// TIA Portal V17 program export: 11 tag tables, 0 data types, 34 data blocks, 53 code blocks (in call order from the OBs), 52 instance data blocks

VAR_GLOBAL   // PLC tag table "Default tag table"
END_VAR

VAR_GLOBAL   // PLC tag table "St0_In"
   IO_AU_1 AT %I0.0 : Bool;   // Arrêt d'urgence n°1
   IO_AU_2 AT %I0.1 : Bool;   // Arrêt d'urgence n°2
   IO_BP_Rearm AT %I0.2 : Bool;   // Réarmement machine
   IO_Barillet_MP AT %I0.3 : Bool;   // Barillet Métaux Précieux ouvert (MP)
   IO_PorteEntree_Fermee AT %I0.4 : Bool;   // Porte d'entrée : Fermée
   IO_PorteSortie_Fermee AT %I0.5 : Bool;   // Porte de sortie : Fermée
   IO_PorteVision_Fermee AT %I0.6 : Bool;   // Porte maintenance vision façade : Fermée
   IO_PorteArriere_Fermee AT %I0.7 : Bool;   // Portes maitenance arrière machine : Fermée
END_VAR

VAR_GLOBAL   // PLC tag table "St0_Out"
   IO_Verrou_PorteEntree AT %Q0.0 : Bool;   // Verrouillage : Porte d'entrée
   IO_Verrou_PorteSortie AT %Q0.1 : Bool;   // Verrouillage : Porte de sortie
   IO_Verrou_PorteVision AT %Q0.2 : Bool;   // Verrouillage : Porte maintenance vision façade
   IO_Verrou_PorteArriere AT %Q0.3 : Bool;   // Verrouillage : Porte maintenance arrière machine
   IO_Ouverture_PorteEntree AT %Q0.4 : Bool;   // Ouverture : Porte d'entrée
   IO_Ouverture_PorteSortie AT %Q0.5 : Bool;   // Ouverture : Porte de sortie
   IO_LED_Rouge AT %Q0.6 : Bool;   // Colonne lumineuse : Rouge
   IO_LED_Orange AT %Q0.7 : Bool;   // Colonne lumineuse : Orange
   IO_LED_Vert AT %Q1.0 : Bool;   // Colonne lumineuse : Vert
   IO_LED_Bleu AT %Q1.1 : Bool;   // Colonne lumineuse : Bleu
END_VAR

VAR_GLOBAL   // PLC tag table "St1_In"
   IO_Pinces_Ouvert AT %I1.0 : Bool;   // Pinces de préhension Z : Ouverte
   IO_Pinces_Fermee AT %I1.1 : Bool;   // Pinces de préhension Z : Fermée
   IO_Cpt_C1 AT %I1.2 : Bool;   // Présence pile devant capteur Chargement AR : C1
   IO_Cpt_C2 AT %I1.3 : Bool;   // Présence pile devant capteur Chargement AR : C2
   IO_Cpt_C3 AT %I1.4 : Bool;   // Présence pile devant capteur Chargement AV : C3
   IO_Cpt_C4 AT %I1.5 : Bool;   // Présence pile devant capteur Chargement AV : C4
   IO_Cpt_C5 AT %I1.6 : Bool;   // Présence pile devant capteur Dépilement : C5
   IO_Cpt_C6 AT %I1.7 : Bool;   // Détection collage barquette Dépilement : C6
   IO_Cpt_C7 AT %I2.0 : Bool;   // Détection collage barquette Dépilement : C7
END_VAR

VAR_GLOBAL   // PLC tag table "St1_Out"
   IO_Ouverture_Pinces AT %Q1.2 : Bool;   // Ouverture : Pinces de préhension
   IO_Fermeture_Pinces AT %Q1.3 : Bool;   // Fermeture : Pinces de préhension
   IO_Vy_PileAV AT %Q1.4 : Bool;   // Conditions sur voyant C2 : OK
   IO_Vy_PileAR AT %Q1.5 : Bool;   // Conditions sur voyant C4 : OK
END_VAR

VAR_GLOBAL   // PLC tag table "St2_In"
   IO_Cpt_V1 AT %I2.1 : Bool;   // Présence barquette en début de Vision : V1
   IO_Cpt_V2 AT %I2.2 : Bool;   // Détection butée à came : V2
   IO_Cpt_V3 AT %I2.3 : Bool;   // Détection butée pivot : V3
END_VAR

VAR_GLOBAL   // PLC tag table "St2_Out"
END_VAR

VAR_GLOBAL   // PLC tag table "St3_In"
   IO_TrappeEntree_Ouvert AT %I2.4 : Bool;   // Trappe d'entrée : Ouverte
   IO_TrappeEntree_Fermee AT %I2.5 : Bool;   // Trappe d'entrée : Fermée
   IO_TrappeSortie_Ouvert AT %I2.6 : Bool;   // Trappe de sortie : Ouverte
   IO_TrappeSortie_Fermee AT %I2.7 : Bool;   // Trappe de sortie : Fermée
   IO_Obturateur_Ouvert AT %I3.0 : Bool;   // Obturateur : Ouvert
   IO_Obturateur_Fermee AT %I3.1 : Bool;   // Obturateur : Fermé
   IO_PorteRX_Ouvert AT %I3.2 : Bool;   // Porte RX : Ouverte (Homme)
   IO_PorteRX_Fermee AT %I3.3 : Bool;   // Porte RX : Ferméee (Homme)
   IO_Cpt_RX1 AT %I3.4 : Bool;   // Présence barquette en début de RX : RX1
   IO_Cpt_RX2 AT %I3.5 : Bool;   // Détection butée à came : RX2
   IO_Cpt_RX3 AT %I3.6 : Bool;   // Détection butée pivot : RX3
   IO_Vy_Orange AT %I3.7 : Bool;   // Obturateur Fermée + RX Actif
   IO_Vy_Rouge AT %I4.0 : Bool;   // Obturateur Ouvert + RX Actif
END_VAR

VAR_GLOBAL   // PLC tag table "St3_Out"
   IO_Ouverture_TrappeEntree AT %Q1.6 : Bool;   // Ouverture : Trappe d'entrée
   IO_Fermeture_TrappeEntree AT %Q1.7 : Bool;   // Fermeture : Trappe de sortie
   IO_Ouverture_TrappeSortie AT %Q2.0 : Bool;   // Ouverture : Trappe de sortie
   IO_Fermeture_TrappeSortie AT %Q2.1 : Bool;   // Fermeture : Trappe de sortie
   IO_Ouverture_Obturateur AT %Q2.2 : Bool;   // Ouverture : Obturateur
   IO_Fermeture_Obturateur AT %Q2.3 : Bool;   // Fermeture : Obturateur
   IO_Femerture_PorteRX AT %Q2.4 : Bool;   // Ouverte : Porte RX (Homme)
   IO_Ouverture_PorteRX AT %Q2.5 : Bool;   // Fermeture : Porte RX (Homme)
END_VAR

VAR_GLOBAL   // PLC tag table "St4_In"
   IO_Loquet_Haut AT %I4.1 : Bool;   // Loquet haut : Pas de déplacement barquette
   IO_Cpt_M AT %I4.2 : Bool;   // Présence pile en zone de marquage
   IO_PincesDC_Ouvert AT %I4.3 : Bool;   // Pinces de préhension Déchagement C : Ouverte
   IO_PincesDC_Fermee AT %I4.4 : Bool;   // Pinces de préhension Déchagement C : Fermée
   IO_Cpt_DC1 AT %I4.5 : Bool;   // Présence pile en zone Déchagement C1
   IO_Cpt_DC2 AT %I4.6 : Bool;   // Présence pile en zone Déchagement : C2
   IO_PoussoirC_Haut AT %I4.7 : Bool;   // Poussoir C en position : Haut
   IO_PincesDNC_Ouvert AT %I5.0 : Bool;   // Pinces de préhension Déchagement NC : Ouverte
   IO_PincesDNC_Fermee AT %I5.1 : Bool;   // Pinces de préhension Déchagement NC : Ferméee
   IO_Cpt_DNC0 AT %I5.2 : Bool;   // Présence pile en zone Déchagement NC0
   IO_Cpt_DNC1 AT %I5.3 : Bool;   // Présence pile en zone Déchagement DNC1
   IO_Cpt_DNC2 AT %I5.4 : Bool;   // Présence pile en zone Déchagement DNC2
   IO_PoussoirNC_Haut AT %I5.5 : Bool;   // Poussoir NC en position : Haut
END_VAR

VAR_GLOBAL   // PLC tag table "St4_Out"
   IO_Sortir_Loquet AT %Q2.6 : Bool;   // Sortir : Loquet (Déplacement Barquette)
   IO_Sortir_PoussoirC AT %Q2.7 : Bool;   // Sortir : Poussoir Z-OK
   IO_Ouverture_PincesC AT %Q3.0 : Bool;   // Ouverture : Pinces C
   IO_Fermeture_PincesC AT %Q3.1 : Bool;   // Fermeture : Pinces C
   IO_Vy_C AT %Q3.2 : Bool;   // Zone Conforme pleine - A vidanger
   IO_Sortir_PoussoirNC AT %Q3.3 : Bool;   // Sortir Poussoir NC
   IO_Ouverture_PincesNC AT %Q3.4 : Bool;   // Ouverture Pinces NC
   IO_Fermeture_PincesNC AT %Q3.5 : Bool;   // Fermeture Pinces NC
   IO_Vy_NC AT %Q3.6 : Bool;   // Zone Non-Conforme pleine - A vidanger
END_VAR

DATA_BLOCK "Visu"   // DB85
{ S7_Optimized_Access := 'TRUE' }
VERSION : 0.1
// stored: AutoNumber false, DBAccessibleFromOPCUA true, DBAccessibleFromWebserver true, IsOnlyStoredInLoadMemory false, IsRetainMemResEnabled false, IsWriteProtectedInAS false, MemoryReserve 100
   VAR
      Page : Struct
         xAuto : Bool;
         xManu : Bool;
         xPaP : Bool;
      END_STRUCT;
      Pop_Up : Struct
         Open : Bool;
         Close : Bool;
         xOk : Bool;
         xYes : Bool;
         xNo : Bool;
      END_STRUCT;
   END_VAR
BEGIN
END_DATA_BLOCK

DATA_BLOCK "St0_In"   // DB5
{ S7_Optimized_Access := 'TRUE' }
VERSION : 0.1
// stored: AutoNumber false, DBAccessibleFromOPCUA true, DBAccessibleFromWebserver true, IsOnlyStoredInLoadMemory false, IsRetainMemResEnabled false, IsWriteProtectedInAS false, MemoryReserve 100
   VAR
      AU_1 : Bool;   // Arrêt d'urgence n°1
      AU_2 : Bool;   // Arrêt d'urgence n°2
      BP_Rearm : Bool;   // Réarmement machine
      Barillet_MP : Bool;   // Barillet Métaux Précieux ouvert (MP)
      PorteEntree_Fermee : Bool;   // Porte d'entrée : Fermée
      PorteSortie_Fermee : Bool;   // Porte de sortie : Fermée
      PorteVision_Fermee : Bool;   // Porte maintenance vision façade : Fermée
      PorteArriere_Fermee : Bool;   // Portes maitenance arrière machine : Fermée
   END_VAR
BEGIN
END_DATA_BLOCK

DATA_BLOCK "St0_Out"   // DB15
{ S7_Optimized_Access := 'TRUE' }
VERSION : 0.1
// stored: AutoNumber false, DBAccessibleFromOPCUA true, DBAccessibleFromWebserver true, IsOnlyStoredInLoadMemory false, IsRetainMemResEnabled false, IsWriteProtectedInAS false, MemoryReserve 100
   VAR
      Verrou_PorteEntree : Bool;
      Verrou_PorteSortie : Bool;
      Verrou_PorteVision : Bool;
      Verrou_PorteArriere : Bool;
      Ouverture_PorteEntree : Bool;
      Ouverture_PorteSortie : Bool;
      LED_Rouge : Bool;
      LED_Orange : Bool;
      LED_Vert : Bool;
      LED_Bleu : Bool;
   END_VAR
BEGIN
END_DATA_BLOCK

DATA_BLOCK "St0_Mem"   // DB25
{ S7_Optimized_Access := 'TRUE' }
VERSION : 0.1
// stored: AutoNumber false, DBAccessibleFromOPCUA true, DBAccessibleFromWebserver true, IsOnlyStoredInLoadMemory false, IsRetainMemResEnabled false, IsWriteProtectedInAS false, MemoryReserve 100
   VAR
      FM_Metal : Bool;
      FM_Noir : Bool;
      FM_Position : Bool;
   END_VAR
BEGIN
END_DATA_BLOCK

DATA_BLOCK "St0_Obj"   // DB35
{ S7_Optimized_Access := 'TRUE' }
VERSION : 0.1
// stored: AutoNumber false, DBAccessibleFromOPCUA true, DBAccessibleFromWebserver true, IsOnlyStoredInLoadMemory false, IsRetainMemResEnabled false, IsWriteProtectedInAS false, MemoryReserve 100
BEGIN
END_DATA_BLOCK

DATA_BLOCK "St0_Const"   // DB45
{ S7_Optimized_Access := 'TRUE' }
VERSION : 0.1
// stored: AutoNumber false, DBAccessibleFromOPCUA true, DBAccessibleFromWebserver true, IsOnlyStoredInLoadMemory false, IsRetainMemResEnabled false, IsWriteProtectedInAS false, MemoryReserve 100
BEGIN
END_DATA_BLOCK

DATA_BLOCK "St0_Per"   // DB55
{ S7_Optimized_Access := 'TRUE' }
VERSION : 0.1
// stored: AutoNumber false, DBAccessibleFromOPCUA true, DBAccessibleFromWebserver true, IsOnlyStoredInLoadMemory false, IsRetainMemResEnabled false, IsWriteProtectedInAS false, MemoryReserve 100
   VAR RETAIN
      HWID : Struct
         _St1_Axe_X : HW_IO := 279;
         _St1_Axe_Y : HW_IO := 281;
         _St1_Prehenseur_Z : HW_IO := 291;
         _St2_Axe_X1 : HW_IO := 293;
         _St2_Axe_X2 : HW_IO := 303;
         _St2_Prehenseur_Z : HW_IO := 305;
         _St3_Axe_X1 : HW_IO := 315;
         _St3_Axe_X2 : HW_IO := 317;
         _St3_Axe_Y : HW_IO := 327;
         "_St3.Axe_Z" : HW_IO := 387;
         _St4_Axe_X1 : HW_IO := 329;
         _St4_Axe_Y1 : HW_IO := 339;
         _St4_Axe_Y2 : HW_IO := 341;
         _St4_Prehenseur_Z2 : HW_IO := 351;
         _St4_Prehenseur_Z3 : HW_IO := 353;
      END_STRUCT;
   END_VAR
BEGIN
END_DATA_BLOCK

DATA_BLOCK "St0_Var"   // DB65
{ S7_Optimized_Access := 'TRUE' }
VERSION : 0.1
// stored: AutoNumber false, DBAccessibleFromOPCUA true, DBAccessibleFromWebserver true, IsOnlyStoredInLoadMemory false, IsRetainMemResEnabled false, IsWriteProtectedInAS false, MemoryReserve 100
   VAR
      xPaP : Bool;
   END_VAR
BEGIN
END_DATA_BLOCK

DATA_BLOCK "St1_In"   // DB105
{ S7_Optimized_Access := 'TRUE' }
VERSION : 0.1
// stored: AutoNumber false, DBAccessibleFromOPCUA true, DBAccessibleFromWebserver true, IsOnlyStoredInLoadMemory false, IsRetainMemResEnabled false, IsWriteProtectedInAS false, MemoryReserve 100
   VAR
      Pinces_Ouvert : Bool;   // Pinces de préhension Z : Ouverte
      Pinces_Fermee : Bool;   // Pinces de préhension Z : Fermée
      Cpt_C1 : Bool;   // Présence pile devant capteur Chargement AR : C1
      Cpt_C2 : Bool;   // Présence pile devant capteur Chargement AR : C2
      Cpt_C3 : Bool;   // Présence pile devant capteur Chargement AV : C3
      Cpt_C4 : Bool;   // Présence pile devant capteur Chargement AV : C4
      Cpt_C5 : Bool;   // Présence pile devant capteur Dépilement : C5
      Cpt_C6 : Bool;   // Détection collage barquette Dépilement : C6
      Cpt_C7 : Bool;   // Détection collage barquette Dépilement : C7
   END_VAR
BEGIN
END_DATA_BLOCK

DATA_BLOCK "St1_Out"   // DB115
{ S7_Optimized_Access := 'TRUE' }
VERSION : 0.1
// stored: AutoNumber false, DBAccessibleFromOPCUA true, DBAccessibleFromWebserver true, IsOnlyStoredInLoadMemory false, IsRetainMemResEnabled false, IsWriteProtectedInAS false, MemoryReserve 100
   VAR
      Ouverture_Pinces : Bool;   // Ouverture : Pinces de préhension
      Fermeture_Pinces : Bool;   // Fermeture : Pinces de préhension
      Vy_PileAV : Bool;   // Conditions sur voyant C2 : OK
      Vy_PileAR : Bool;   // Conditions sur voyant C4 : OK
   END_VAR
BEGIN
END_DATA_BLOCK

DATA_BLOCK "St1_Mem"   // DB125
{ S7_Optimized_Access := 'TRUE' }
VERSION : 0.1
// stored: AutoNumber false, DBAccessibleFromOPCUA true, DBAccessibleFromWebserver true, IsOnlyStoredInLoadMemory false, IsRetainMemResEnabled false, IsWriteProtectedInAS false, MemoryReserve 100
BEGIN
END_DATA_BLOCK

DATA_BLOCK "St1_Const"   // DB145
{ S7_Optimized_Access := 'TRUE' }
VERSION : 0.1
// stored: AutoNumber false, DBAccessibleFromOPCUA true, DBAccessibleFromWebserver true, IsOnlyStoredInLoadMemory false, IsRetainMemResEnabled false, IsWriteProtectedInAS false, MemoryReserve 100
BEGIN
END_DATA_BLOCK

DATA_BLOCK "St1_Per"   // DB155
{ S7_Optimized_Access := 'TRUE' }
VERSION : 0.1
// stored: AutoNumber false, DBAccessibleFromOPCUA true, DBAccessibleFromWebserver true, IsOnlyStoredInLoadMemory false, IsRetainMemResEnabled false, IsWriteProtectedInAS false, MemoryReserve 100
BEGIN
END_DATA_BLOCK

DATA_BLOCK "St1_Var"   // DB165
{ S7_Optimized_Access := 'TRUE' }
VERSION : 0.1
// stored: AutoNumber false, DBAccessibleFromOPCUA true, DBAccessibleFromWebserver true, IsOnlyStoredInLoadMemory false, IsRetainMemResEnabled false, IsWriteProtectedInAS false, MemoryReserve 100
BEGIN
END_DATA_BLOCK

DATA_BLOCK "St2_In"   // DB205
{ S7_Optimized_Access := 'TRUE' }
VERSION : 0.1
// stored: AutoNumber false, DBAccessibleFromOPCUA true, DBAccessibleFromWebserver true, IsOnlyStoredInLoadMemory false, IsRetainMemResEnabled false, IsWriteProtectedInAS false, MemoryReserve 100
   VAR
      Cpt_V1 : Bool;   // Présence barquette en début de Vision : V1
      Cpt_V2 : Bool;   // Détection butée à came : V2
      Cpt_V3 : Bool;   // Détection butée pivot : V3
   END_VAR
BEGIN
END_DATA_BLOCK

DATA_BLOCK "St2_Out"   // DB215
{ S7_Optimized_Access := 'TRUE' }
VERSION : 0.1
// stored: AutoNumber false, DBAccessibleFromOPCUA true, DBAccessibleFromWebserver true, IsOnlyStoredInLoadMemory false, IsRetainMemResEnabled false, IsWriteProtectedInAS false, MemoryReserve 100
BEGIN
END_DATA_BLOCK

DATA_BLOCK "St2_Mem"   // DB225
{ S7_Optimized_Access := 'TRUE' }
VERSION : 0.1
// stored: AutoNumber false, DBAccessibleFromOPCUA true, DBAccessibleFromWebserver true, IsOnlyStoredInLoadMemory false, IsRetainMemResEnabled false, IsWriteProtectedInAS false, MemoryReserve 100
   VAR
      FM_Metal : Bool;
      FM_Noir : Bool;
      FM_Position : Bool;
   END_VAR
BEGIN
END_DATA_BLOCK

DATA_BLOCK "St2_Const"   // DB245
{ S7_Optimized_Access := 'TRUE' }
VERSION : 0.1
// stored: AutoNumber false, DBAccessibleFromOPCUA true, DBAccessibleFromWebserver true, IsOnlyStoredInLoadMemory false, IsRetainMemResEnabled false, IsWriteProtectedInAS false, MemoryReserve 100
BEGIN
END_DATA_BLOCK

DATA_BLOCK "St2_Per"   // DB255
{ S7_Optimized_Access := 'TRUE' }
VERSION : 0.1
// stored: AutoNumber false, DBAccessibleFromOPCUA true, DBAccessibleFromWebserver true, IsOnlyStoredInLoadMemory false, IsRetainMemResEnabled false, IsWriteProtectedInAS false, MemoryReserve 100
BEGIN
END_DATA_BLOCK

DATA_BLOCK "St2_Var"   // DB265
{ S7_Optimized_Access := 'TRUE' }
VERSION : 0.1
// stored: AutoNumber false, DBAccessibleFromOPCUA true, DBAccessibleFromWebserver true, IsOnlyStoredInLoadMemory false, IsRetainMemResEnabled false, IsWriteProtectedInAS false, MemoryReserve 100
   VAR
      Fin_Vision : Bool;
   END_VAR
BEGIN
END_DATA_BLOCK

DATA_BLOCK "St3_In"   // DB305
{ S7_Optimized_Access := 'TRUE' }
VERSION : 0.1
// stored: AutoNumber false, DBAccessibleFromOPCUA true, DBAccessibleFromWebserver true, IsOnlyStoredInLoadMemory false, IsRetainMemResEnabled false, IsWriteProtectedInAS false, MemoryReserve 100
   VAR
      TrappeEntree_Ouvert : Bool;   // Trappe d'entrée : Ouverte
      TrappeEntree_Fermee : Bool;   // Trappe d'entrée : Fermée
      TrappeSortie_Ouvert : Bool;   // Trappe de sortie : Ouverte
      TrappeSortie_Fermee : Bool;   // Trappe de sortie : Fermée
      Obturateur_Ouvert : Bool;   // Obturateur : Ouvert
      Obturateur_Fermee : Bool;   // Obturateur : Fermé
      PorteRX_Ouvert : Bool;   // Porte RX : Ouverte (Homme)
      PorteRX_Fermee : Bool;   // Porte RX : Ferméee (Homme)
      Cpt_RX1 : Bool;   // Présence barquette en début de RX : RX1
      Cpt_RX2 : Bool;   // Détection butée à came : RX2
      Cpt_RX3 : Bool;   // Détection butée pivot : RX3
      Vy_Orange : Bool;   // Obturateur Fermée + RX Actif
      Vy_Rouge : Bool;   // Obturateur Ouvert + RX Actif
   END_VAR
BEGIN
END_DATA_BLOCK

DATA_BLOCK "St3_Out"   // DB315
{ S7_Optimized_Access := 'TRUE' }
VERSION : 0.1
// stored: AutoNumber false, DBAccessibleFromOPCUA true, DBAccessibleFromWebserver true, IsOnlyStoredInLoadMemory false, IsRetainMemResEnabled false, IsWriteProtectedInAS false, MemoryReserve 100
   VAR
      Ouverture_TrappeEntree : Bool;   // Ouverture : Trappe d'entrée
      Fermeture_TrappeEntree : Bool;   // Fermeture : Trappe de sortie
      Ouverture_TrappeSortie : Bool;   // Ouverture : Trappe de sortie
      Fermeture_TrappeSortie : Bool;   // Fermeture : Trappe de sortie
      Ouverture_Obturateur : Bool;   // Ouverture : Obturateur
      Fermeture_Obturateur : Bool;   // Fermeture : Obturateur
      Femerture_PorteRX : Bool;   // Ouverte : Porte RX (Homme)
      Ouverture_PorteRX : Bool;   // Fermeture : Porte RX (Homme)
   END_VAR
BEGIN
END_DATA_BLOCK

DATA_BLOCK "St3_Mem"   // DB325
{ S7_Optimized_Access := 'TRUE' }
VERSION : 0.1
// stored: AutoNumber false, DBAccessibleFromOPCUA true, DBAccessibleFromWebserver true, IsOnlyStoredInLoadMemory false, IsRetainMemResEnabled false, IsWriteProtectedInAS false, MemoryReserve 100
   VAR
      FM_Metal : Bool;
      FM_Noir : Bool;
      FM_Position : Bool;
   END_VAR
BEGIN
END_DATA_BLOCK

DATA_BLOCK "St3_Const"   // DB345
{ S7_Optimized_Access := 'TRUE' }
VERSION : 0.1
// stored: AutoNumber false, DBAccessibleFromOPCUA true, DBAccessibleFromWebserver true, IsOnlyStoredInLoadMemory false, IsRetainMemResEnabled false, IsWriteProtectedInAS false, MemoryReserve 100
BEGIN
END_DATA_BLOCK

DATA_BLOCK "St3_Per"   // DB355
{ S7_Optimized_Access := 'TRUE' }
VERSION : 0.1
// stored: AutoNumber false, DBAccessibleFromOPCUA true, DBAccessibleFromWebserver true, IsOnlyStoredInLoadMemory false, IsRetainMemResEnabled false, IsWriteProtectedInAS false, MemoryReserve 100
BEGIN
END_DATA_BLOCK

DATA_BLOCK "St3_Var"   // DB365
{ S7_Optimized_Access := 'TRUE' }
VERSION : 0.1
// stored: AutoNumber false, DBAccessibleFromOPCUA true, DBAccessibleFromWebserver true, IsOnlyStoredInLoadMemory false, IsRetainMemResEnabled false, IsWriteProtectedInAS false, MemoryReserve 100
BEGIN
END_DATA_BLOCK

DATA_BLOCK "St4_In"   // DB405
{ S7_Optimized_Access := 'TRUE' }
VERSION : 0.1
// stored: AutoNumber false, DBAccessibleFromOPCUA true, DBAccessibleFromWebserver true, IsOnlyStoredInLoadMemory false, IsRetainMemResEnabled false, IsWriteProtectedInAS false, MemoryReserve 100
   VAR
      Loquet_Haut : Bool;   // Loquet haut : Pas de déplacement barquette
      Cpt_M : Bool;   // Présence pile en zone de marquage
      PincesDC_Ouvert : Bool;   // Pinces de préhension Déchagement C : Ouverte
      PincesDC_Fermee : Bool;   // Pinces de préhension Déchagement C : Fermée
      Cpt_DC1 : Bool;   // Présence pile en zone Déchagement C1
      Cpt_DC2 : Bool;   // Présence pile en zone Déchagement : C2
      PoussoirC_Haut : Bool;   // Poussoir C en position : Haut
      PincesDNC_Ouvert : Bool;   // Pinces de préhension Déchagement NC : Ouverte
      PincesDNC_Fermee : Bool;   // Pinces de préhension Déchagement NC : Ferméee
      Cpt_DNC0 : Bool;   // Présence pile en zone Déchagement NC0
      Cpt_DNC1 : Bool;   // Présence pile en zone Déchagement DNC1
      Cpt_DNC2 : Bool;   // Présence pile en zone Déchagement DNC2
      PoussoirNC_Haut : Bool;   // Poussoir NC en position : Haut
   END_VAR
BEGIN
END_DATA_BLOCK

DATA_BLOCK "St4_Out"   // DB415
{ S7_Optimized_Access := 'TRUE' }
VERSION : 0.1
// stored: AutoNumber false, DBAccessibleFromOPCUA true, DBAccessibleFromWebserver true, IsOnlyStoredInLoadMemory false, IsRetainMemResEnabled false, IsWriteProtectedInAS false, MemoryReserve 100
   VAR
      Sortir_Loquet : Bool;   // Sortir : Loquet (Déplacement Barquette)
      Sortir_PoussoirC : Bool;   // Sortir : Poussoir Z-OK
      Ouverture_PincesC : Bool;   // Ouverture : Pinces C
      Fermeture_PincesC : Bool;   // Fermeture : Pinces C
      Vy_C : Bool;   // Zone Conforme pleine - A vidanger
      Sortir_PoussoirNC : Bool;   // Sortir Poussoir NC
      Ouverture_PincesNC : Bool;   // Ouverture Pinces NC
      Fermeture_PincesNC : Bool;   // Fermeture Pinces NC
      Vy_NC : Bool;   // Zone Non-Conforme pleine - A vidanger
   END_VAR
BEGIN
END_DATA_BLOCK

DATA_BLOCK "St4_Mem"   // DB425
{ S7_Optimized_Access := 'TRUE' }
VERSION : 0.1
// stored: AutoNumber false, DBAccessibleFromOPCUA true, DBAccessibleFromWebserver true, IsOnlyStoredInLoadMemory false, IsRetainMemResEnabled false, IsWriteProtectedInAS false, MemoryReserve 100
   VAR
      FM_Metal : Bool;
      FM_Noir : Bool;
      FM_Position : Bool;
   END_VAR
BEGIN
END_DATA_BLOCK

DATA_BLOCK "St4_Const"   // DB445
{ S7_Optimized_Access := 'TRUE' }
VERSION : 0.1
// stored: AutoNumber false, DBAccessibleFromOPCUA true, DBAccessibleFromWebserver true, IsOnlyStoredInLoadMemory false, IsRetainMemResEnabled false, IsWriteProtectedInAS false, MemoryReserve 100
BEGIN
END_DATA_BLOCK

DATA_BLOCK "St4_Per"   // DB455
{ S7_Optimized_Access := 'TRUE' }
VERSION : 0.1
// stored: AutoNumber false, DBAccessibleFromOPCUA true, DBAccessibleFromWebserver true, IsOnlyStoredInLoadMemory false, IsRetainMemResEnabled false, IsWriteProtectedInAS false, MemoryReserve 100
BEGIN
END_DATA_BLOCK

DATA_BLOCK "St4_Var"   // DB465
{ S7_Optimized_Access := 'TRUE' }
VERSION : 0.1
// stored: AutoNumber false, DBAccessibleFromOPCUA true, DBAccessibleFromWebserver true, IsOnlyStoredInLoadMemory false, IsRetainMemResEnabled false, IsWriteProtectedInAS false, MemoryReserve 100
BEGIN
END_DATA_BLOCK

DATA_BLOCK "RCT"   // DB1005
{ S7_Optimized_Access := 'TRUE' }
VERSION : 0.1
// stored: AutoNumber false, DBAccessibleFromOPCUA true, DBAccessibleFromWebserver true, IsOnlyStoredInLoadMemory false, IsRetainMemResEnabled false, IsWriteProtectedInAS false, MemoryReserve 100
   VAR
      St2 : Struct
         Axe_X1 : Struct
            Vel_Vision : LReal;
            Pos_Vision : LReal;
            ModeAbs : Bool;
            ModeRel : Bool;
         END_STRUCT;
         Prehenseur_Z : Struct
            Pos_Vision : LReal;
         END_STRUCT;
         Autorisation_Vision : Bool;
         Fin_Vision : Bool;
      END_STRUCT;
      St3 : Struct
         Axe_X1 : Struct
            Vel_RX : LReal;
            Pos_RX : LReal;
            ModeAbs : Bool;
            ModeRel : Bool;
         END_STRUCT;
         Axe_Y : Struct
            Pos_RX : LReal;
         END_STRUCT;
         Axe_Z : Struct
            Pos_RX : LReal;
         END_STRUCT;
         Autorisation_RX : Bool;
         Fin_RX : Bool;
      END_STRUCT;
      St4 : Struct
         Axe_X1 : Struct
            Pos_Marquage : LReal;
         END_STRUCT;
         Axe_Y1 : Struct
            Pos_Marquage : LReal;
         END_STRUCT;
      END_STRUCT;
   END_VAR
BEGIN
END_DATA_BLOCK

DATA_BLOCK "OF"   // DB1015
{ S7_Optimized_Access := 'TRUE' }
VERSION : 0.1
// stored: AutoNumber false, DBAccessibleFromOPCUA true, DBAccessibleFromWebserver true, IsOnlyStoredInLoadMemory false, IsRetainMemResEnabled false, IsWriteProtectedInAS false, MemoryReserve 100
BEGIN
END_DATA_BLOCK

ORGANIZATION_BLOCK "Main"   // OB1, LAD, ProgramCycle
TITLE = "Main Program Sweep (Cycle)"
{ S7_Optimized_Access := 'TRUE' }
VERSION : 0.1
// *********************  Création : 01/06/2024  *********************
// *****************  Kep Technologies - Caluire 69150  ****************
// ************************  RM Automation  ***********************
// **********************  Auteur: Rebouh.M  ***********************
// ***************** Contact : Rebouh.mehdi@hotmail.fr  ***************
// stored: AutoNumber true, IsIECCheckEnabled false, SetENOAutomatically false
   VAR_INPUT
      Initial_Call : Bool;   // Initial call of this OB
      Remanence : Bool;   // =True, if remanent data are available
   END_VAR
BEGIN

REGION Network 1: Manager
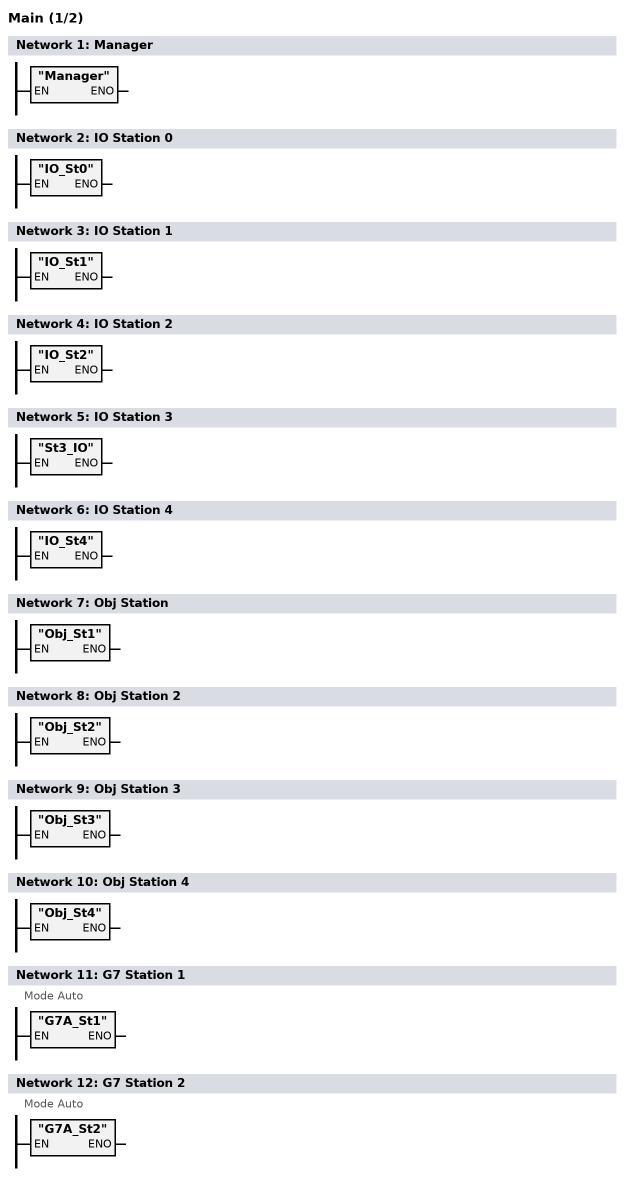
   RUNG wire#powerrail
      "Manager"()
   END_RUNG
   // the same network as SCL:
   "Manager"();
END_REGION

REGION Network 2: IO Station 0
   RUNG wire#powerrail
      "IO_St0"()
   END_RUNG
   // the same network as SCL:
   "IO_St0"();
END_REGION

REGION Network 3: IO Station 1
   RUNG wire#powerrail
      "IO_St1"()
   END_RUNG
   // the same network as SCL:
   "IO_St1"();
END_REGION

REGION Network 4: IO Station 2
   RUNG wire#powerrail
      "IO_St2"()
   END_RUNG
   // the same network as SCL:
   "IO_St2"();
END_REGION

REGION Network 5: IO Station 3
   RUNG wire#powerrail
      "St3_IO"()
   END_RUNG
   // the same network as SCL:
   "St3_IO"();
END_REGION

REGION Network 6: IO Station 4
   RUNG wire#powerrail
      "IO_St4"()
   END_RUNG
   // the same network as SCL:
   "IO_St4"();
END_REGION

REGION Network 7: Obj Station
   RUNG wire#powerrail
      "Obj_St1"()
   END_RUNG
   // the same network as SCL:
   "Obj_St1"();
END_REGION

REGION Network 8: Obj Station 2
   RUNG wire#powerrail
      "Obj_St2"()
   END_RUNG
   // the same network as SCL:
   "Obj_St2"();
END_REGION

REGION Network 9: Obj Station 3
   RUNG wire#powerrail
      "Obj_St3"()
   END_RUNG
   // the same network as SCL:
   "Obj_St3"();
END_REGION

REGION Network 10: Obj Station 4
   RUNG wire#powerrail
      "Obj_St4"()
   END_RUNG
   // the same network as SCL:
   "Obj_St4"();
END_REGION

REGION Network 11: G7 Station 1
   // Mode Auto
   RUNG wire#powerrail
      "G7A_St1"()
   END_RUNG
   // the same network as SCL:
   "G7A_St1"();
END_REGION

REGION Network 12: G7 Station 2
   // Mode Auto
   RUNG wire#powerrail
      "G7A_St2"()
   END_RUNG
   // the same network as SCL:
   "G7A_St2"();
END_REGION

REGION Network 13: G7 Station 3
   // Mode Auto
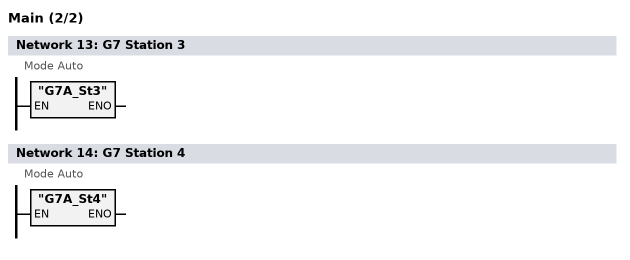
   RUNG wire#powerrail
      "G7A_St3"()
   END_RUNG
   // the same network as SCL:
   "G7A_St3"();
END_REGION

REGION Network 14: G7 Station 4
   // Mode Auto
   RUNG wire#powerrail
      "G7A_St4"()
   END_RUNG
   // the same network as SCL:
   "G7A_St4"();
END_REGION
END_ORGANIZATION_BLOCK

FUNCTION "Manager" : Void   // FC1, LAD
{ S7_Optimized_Access := 'TRUE' }
VERSION : 0.1
// stored: AutoNumber false, IsIECCheckEnabled false, SetENOAutomatically false, UDAEnableTagReadback false
BEGIN

REGION Network 1
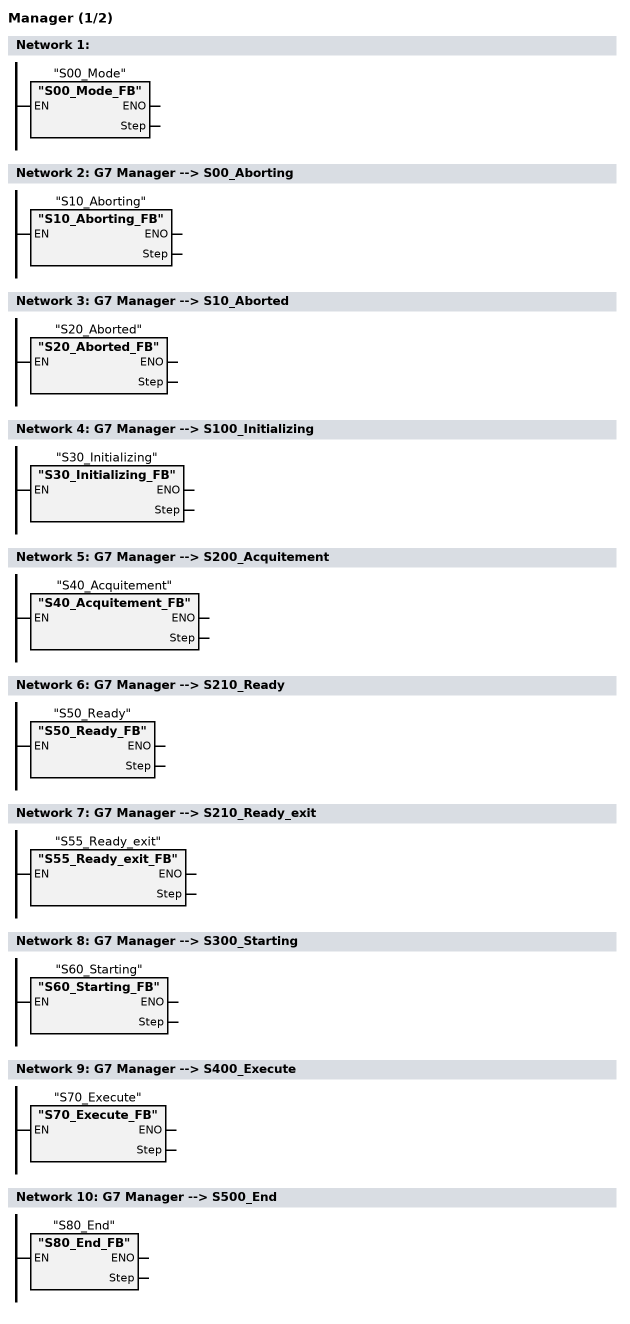
   RUNG wire#powerrail
      "S00_Mode"("Step" =>)
   END_RUNG
   // the same network as SCL:
   "S00_Mode"();   // "S00_Mode_FB"
END_REGION

REGION Network 2: G7 Manager --> S00_Aborting
   RUNG wire#powerrail
      "S10_Aborting"("Step" =>)
   END_RUNG
   // the same network as SCL:
   "S10_Aborting"();   // "S10_Aborting_FB"
END_REGION

REGION Network 3: G7 Manager --> S10_Aborted
   RUNG wire#powerrail
      "S20_Aborted"("Step" =>)
   END_RUNG
   // the same network as SCL:
   "S20_Aborted"();   // "S20_Aborted_FB"
END_REGION

REGION Network 4: G7 Manager --> S100_Initializing
   RUNG wire#powerrail
      "S30_Initializing"("Step" =>)
   END_RUNG
   // the same network as SCL:
   "S30_Initializing"();   // "S30_Initializing_FB"
END_REGION

REGION Network 5: G7 Manager --> S200_Acquitement
   RUNG wire#powerrail
      "S40_Acquitement"("Step" =>)
   END_RUNG
   // the same network as SCL:
   "S40_Acquitement"();   // "S40_Acquitement_FB"
END_REGION

REGION Network 6: G7 Manager --> S210_Ready
   RUNG wire#powerrail
      "S50_Ready"("Step" =>)
   END_RUNG
   // the same network as SCL:
   "S50_Ready"();   // "S50_Ready_FB"
END_REGION

REGION Network 7: G7 Manager --> S210_Ready_exit
   RUNG wire#powerrail
      "S55_Ready_exit"("Step" =>)
   END_RUNG
   // the same network as SCL:
   "S55_Ready_exit"();   // "S55_Ready_exit_FB"
END_REGION

REGION Network 8: G7 Manager --> S300_Starting
   RUNG wire#powerrail
      "S60_Starting"("Step" =>)
   END_RUNG
   // the same network as SCL:
   "S60_Starting"();   // "S60_Starting_FB"
END_REGION

REGION Network 9: G7 Manager --> S400_Execute
   RUNG wire#powerrail
      "S70_Execute"("Step" =>)
   END_RUNG
   // the same network as SCL:
   "S70_Execute"();   // "S70_Execute_FB"
END_REGION

REGION Network 10: G7 Manager --> S500_End
   RUNG wire#powerrail
      "S80_End"("Step" =>)
   END_RUNG
   // the same network as SCL:
   "S80_End"();   // "S80_End_FB"
END_REGION

REGION Network 11: G7 Manager --> S600_Stopping
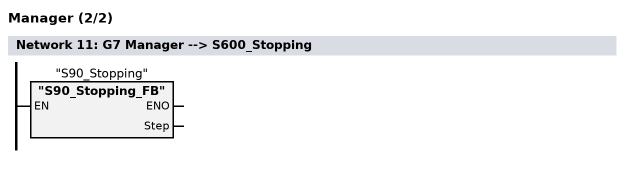
   RUNG wire#powerrail
      "S90_Stopping"("Step" =>)
   END_RUNG
   // the same network as SCL:
   "S90_Stopping"();   // "S90_Stopping_FB"
END_REGION
END_FUNCTION

FUNCTION_BLOCK "S00_Mode_FB"
{ S7_Optimized_Access := 'TRUE' }
VERSION : 0.1
   VAR_OUTPUT 
      Step : Int;
   END_VAR

   VAR 
      Step_100 : Int;
      Auto : Bool;
      Manu : Bool;
      PaP : Bool;
   END_VAR


BEGIN
	                
	                (* Manager : S00_Mode *)
	
	// Etape en cours
	#Step := #Step_100;
	
	CASE #Step_100 OF
	        
	    0 :  // Etape Init
	        #Step_100 := 10;
	        
	        
	    10 : // Choix du mode
	        ////////// AUTO /////////// 
	        IF "Visu".Page.xAuto THEN
	            #Auto := TRUE;
	            #Step_100 := 100;
	        END_IF;
	      ////////// MANU /////////// 
	        IF "Visu".Page.xManu THEN
	            #Manu := TRUE;
	            #Step_100 := 200;
	        END_IF;
	      ////////// PaP /////////// 
	        IF "Visu".Page.xPaP THEN
	            #PaP := TRUE;
	            #Step_100 := 300;
	        END_IF;
	      
	      
	    100 : // OUT AUTO
	        IF NOT "Visu".Page.xAuto THEN
	            #Auto := FALSE;
	            #Step_100 := 10;
	        END_IF;
	        
	        
	    200 : // OUT MANU
	        IF NOT "Visu".Page.xManu THEN
	            #Manu := FALSE;
	            #Step_100 := 10;
	        END_IF;
	        
	        
	    300 : // OUT PAP
	        IF NOT "Visu".Page.xPaP THEN
	            #PaP := FALSE;
	            #Step_100 := 10;
	        END_IF;
	        
	        
	END_CASE;
	
	
END_FUNCTION_BLOCK

FUNCTION_BLOCK "S10_Aborting_FB"
{ S7_Optimized_Access := 'TRUE' }
VERSION : 0.1
   VAR_OUTPUT 
      Step : Int;
   END_VAR

   VAR 
      Step_100 : Int;
   END_VAR


BEGIN
	                
	                (* Manager : S10_Aborting *)
	
	// Etape en cours
	#Step := #Step_100;
	
	CASE #Step_100 OF
	        
	    0:  // Etape Init
	        #Step_100 := 10;
	        
	END_CASE;
END_FUNCTION_BLOCK

FUNCTION_BLOCK "S20_Aborted_FB"
{ S7_Optimized_Access := 'TRUE' }
VERSION : 0.1
   VAR_OUTPUT 
      Step : Int;
   END_VAR

   VAR 
      Step_100 : Int;
   END_VAR


BEGIN
	
	                (* Manager : S20_Aborted *)
	
	// Etape en cours
	#Step := #Step_100;
	
	CASE #Step_100 OF
	        
	    0:  // Etape Init
	        #Step_100 := 10;
	        
	END_CASE;
END_FUNCTION_BLOCK

FUNCTION_BLOCK "S30_Initializing_FB"
{ S7_Optimized_Access := 'TRUE' }
VERSION : 0.1
   VAR_OUTPUT 
      Step : Int;
   END_VAR

   VAR 
      Step_100 : Int;
   END_VAR


BEGIN
	
	                (* Manager : S30_Initializing *)
	
	// Etape en cours
	#Step := #Step_100;
	
	CASE #Step_100 OF
	        
	    0:  // Etape Init
	        #Step_100 := 10;
	        
	END_CASE;
END_FUNCTION_BLOCK

FUNCTION_BLOCK "S40_Acquitement_FB"
{ S7_Optimized_Access := 'TRUE' }
VERSION : 0.1
   VAR_OUTPUT 
      Step : Int;
   END_VAR

   VAR 
      Step_100 : Int;
   END_VAR


BEGIN
	
	                (* Manager : S40_Acquitement *)
	
	// Etape en cours
	#Step := #Step_100;
	
	CASE #Step_100 OF
	        
	    0:  // Etape Init
	        #Step_100 := 10;
	        
	END_CASE;
END_FUNCTION_BLOCK

FUNCTION_BLOCK "S50_Ready_FB"
{ S7_Optimized_Access := 'TRUE' }
VERSION : 0.1
   VAR_OUTPUT 
      Step : Int;
   END_VAR

   VAR 
      Step_100 : Int;
   END_VAR


BEGIN
	
	                (* Manager : S50_Ready *)
	
	// Etape en cours
	#Step := #Step_100;
	
	CASE #Step_100 OF
	        
	    0:  // Etape Init
	        #Step_100 := 10;
	        
	END_CASE;
END_FUNCTION_BLOCK

FUNCTION_BLOCK "S55_Ready_exit_FB"
{ S7_Optimized_Access := 'TRUE' }
VERSION : 0.1
   VAR_OUTPUT 
      Step : Int;
   END_VAR

   VAR 
      Step_100 : Int;
   END_VAR


BEGIN
	
	                (* Manager : S55_Ready_exit *)
	
	// Etape en cours
	#Step := #Step_100;
	
	CASE #Step_100 OF
	        
	    0:  // Etape Init
	        #Step_100 := 10;
	        
	END_CASE;
END_FUNCTION_BLOCK

FUNCTION_BLOCK "S60_Starting_FB"
{ S7_Optimized_Access := 'TRUE' }
VERSION : 0.1
   VAR_OUTPUT 
      Step : Int;
   END_VAR

   VAR 
      Step_100 : Int;
   END_VAR


BEGIN
	
	                (* Manager : S60_Starting *)
	
	// Etape en cours
	#Step := #Step_100;
	
	CASE #Step_100 OF
	        
	    0:  // Etape Init
	        #Step_100 := 10;
	        
	END_CASE;
END_FUNCTION_BLOCK

FUNCTION_BLOCK "S70_Execute_FB"
{ S7_Optimized_Access := 'TRUE' }
VERSION : 0.1
   VAR_OUTPUT 
      Step : Int;
   END_VAR

   VAR 
      Step_100 : Int;
   END_VAR


BEGIN
	
	                (* Manager : S70_Execute *)
	
	// Etape en cours
	#Step := #Step_100;
	
	CASE #Step_100 OF
	        
	    0:  // Etape Init
	        #Step_100 := 10;
	        
	END_CASE;
END_FUNCTION_BLOCK

FUNCTION_BLOCK "S80_End_FB"
{ S7_Optimized_Access := 'TRUE' }
VERSION : 0.1
   VAR_OUTPUT 
      Step : Int;
   END_VAR

   VAR 
      Step_100 : Int;
   END_VAR


BEGIN
	
	                (* Manager : S80_End *)
	
	// Etape en cours
	#Step := #Step_100;
	
	CASE #Step_100 OF
	        
	    0:  // Etape Init
	        #Step_100 := 10;
	        
	END_CASE;
END_FUNCTION_BLOCK

FUNCTION_BLOCK "S90_Stopping_FB"
{ S7_Optimized_Access := 'TRUE' }
VERSION : 0.1
   VAR_OUTPUT 
      Step : Int;
   END_VAR

   VAR 
      Step_100 : Int;
   END_VAR


BEGIN
	
	                (* Manager : S90_Stopping *)
	
	// Etape en cours
	#Step := #Step_100;
	
	CASE #Step_100 OF
	        
	    0:  // Etape Init
	        #Step_100 := 10;
	        
	END_CASE;
END_FUNCTION_BLOCK

FUNCTION "IO_St0" : Void
{ S7_Optimized_Access := 'TRUE' }
VERSION : 0.1

BEGIN
	
	        (* IO - Station 0 : Machine *)
	
	
	                  (* Input *)
	
	    //___ %I0.0 - Arrêt d'urgence n°1
	    "St0_In".AU_1 := "IO_AU_1";
	    
	    //___ %I0.1 - Arrêt d'urgence n°2
	    "St0_In".AU_2 := "IO_AU_2";
	    
	    //___ %I0.2 - Réarmement machine
	    "St0_In".BP_Rearm := "IO_BP_Rearm";
	    
	    //___ %I0.3 - IO_Barillet_MP
	    "St0_In".Barillet_MP := "IO_Barillet_MP";
	    
	    //___ %I0.4 - Porte d'entrée : Fermée 
	    "St0_In".PorteEntree_Fermee := "IO_PorteEntree_Fermee";
	    
	    //___ %I0.5 - Porte de sortie : Fermée
	    "St0_In".PorteSortie_Fermee := "IO_PorteSortie_Fermee";
	    
	    //___ %I0.6 - Porte maintenance vision façade : Fermée
	    "St0_In".PorteVision_Fermee := "IO_PorteVision_Fermee";
	    
	    //___ %I0.7 - Portes maitenance arrière machine : Fermée
	    "St0_In".PorteArriere_Fermee := "IO_PorteArriere_Fermee";
	    
	    
	                   (* Output *)
	    
	    //___ %Q0.0 - Verrouillage : Porte d'entrée
	    "IO_Verrou_PorteEntree" := "St0_Out".Verrou_PorteEntree;
	    
	    //___ %Q0.1 - Verrouillage : Porte de sortie
	    "IO_Verrou_PorteSortie" := "St0_Out".Verrou_PorteSortie;
	    
	    //___ %Q0.2 - Verrouillage : Porte maintenance vision façade
	    "IO_Verrou_PorteVision" := "St0_Out".Verrou_PorteVision;
	    
	    //___ %Q0.3 - Verrouillage : Porte maintenance arrière machine
	    "IO_Verrou_PorteArriere" := "St0_Out".Verrou_PorteArriere;
	    
	    //___ %Q0.4 - Ouverture : Porte d'entrée
	    "IO_Ouverture_PorteEntree" := "St0_Out".Ouverture_PorteEntree;
	    
	    //___ %Q0.5 - Ouverture : Porte de sortie
	    "IO_Ouverture_PorteSortie" := "St0_Out".Ouverture_PorteSortie;
	    
	    //___ %Q0.6 - Colonne lumineuse : Rouge
	    "IO_LED_Rouge" := "St0_Out".LED_Rouge;
	    
	    //___ %Q0.7 - Colonne lumineuse : Orange
	    "IO_LED_Orange" := "St0_Out".LED_Orange;
	    
	    //___ %Q1.0 - Colonne lumineuse : Vert
	    "IO_LED_Vert" := "St0_Out".LED_Vert;
	    
	    //___ %Q1.1 - Colonne lumineuse : Bleu
	    "IO_LED_Bleu" := "St0_Out".LED_Bleu;
	    
	    
END_FUNCTION

FUNCTION "IO_St1" : Void
{ S7_Optimized_Access := 'TRUE' }
VERSION : 0.1

BEGIN
	
	        (* IO - Station 1 : Chargement - Empilement *)
	
	
	                  (* Input *)
	
	    //___ %I1.0 - Pinces de préhension Z : Ouverte
	    "St1_In".Pinces_Ouvert := "IO_Pinces_Ouvert";
	    
	    //___ %I1.1 - Pinces de préhension Z : Fermée
	    "St1_In".Pinces_Fermee := "IO_Pinces_Fermee";
	    
	    //___ %I1.2 - Présence pile devant capteur Chargement AR : C1
	    "St1_In".Cpt_C1 := "IO_Cpt_C1";
	    
	    //___ %I1.3 - Présence pile devant capteur Chargement AR : C2
	    "St1_In".Cpt_C2 := "IO_Cpt_C2";
	    
	    //___ %I1.4 - Présence pile devant capteur Chargement AV : C3
	    "St1_In".Cpt_C3 := "IO_Cpt_C3";
	    
	    //___ %I1.5 - Présence pile devant capteur Chargement AV : C4
	    "St1_In".Cpt_C4 := "IO_Cpt_C4";
	    
	    //___ %I1.6 - Présence pile devant capteur Dépilement : C5
	    "St1_In".Cpt_C5 := "IO_Cpt_C5";
	    
	    //___ %I1.7 - Détection collage barquette Dépilement : C6 
	    "St1_In".Cpt_C6 := "IO_Cpt_C6";
	    
	    //___ %I2.0 - Détection collage barquette Dépilement : C7 
	    "St1_In".Cpt_C7 := "IO_Cpt_C7";
	    
	    
	                   (* Output *)
	    
	    //___ %Q1.2 - Ouverture : Pinces de préhension 
	    "IO_Ouverture_Pinces" := "St1_Out".Ouverture_Pinces;
	    
	    //___ %Q1.3 - Fermeture : Pinces de préhension
	    "IO_Fermeture_Pinces" := "St1_Out".Fermeture_Pinces;
	    
	    //___ %Q1.4 - Conditions sur voyant C2 : OK
	    "IO_Vy_PileAV" := "St1_Out".Vy_PileAV;
	    
	    //___ %Q1.5 - Conditions sur voyant C4 : OK
	    "IO_Vy_PileAR" := "St1_Out".Vy_PileAR;
	    
	    
	    
END_FUNCTION

FUNCTION "IO_St2" : Void
{ S7_Optimized_Access := 'TRUE' }
VERSION : 0.1

BEGIN
	
	        (* IO - Station 2 : Vision *)
	
	
	                  (* Input *)
	
	    //___ %I2.1 - Présence barquette en début de Vision : V1
	    "St2_In".Cpt_V1 := "IO_Cpt_V1";
	    
	    //___ %I2.2 - Détection butée à came : V2
	    "St2_In".Cpt_V2 := "IO_Cpt_V2";
	    
	    //___ %I2.3 - Détection butée pivot : V3
	    "St2_In".Cpt_V3 := "IO_Cpt_V3";
	    
	
	                   (* Output *)
END_FUNCTION

FUNCTION "St3_IO" : Void
{ S7_Optimized_Access := 'TRUE' }
VERSION : 0.1

BEGIN
	
	        (* IO - Station 3 : RX *)
	
	
	                  (* Input *)
	
	    //___ %I2.4 - Trappe d'entrée : Ouverte
	    "St3_In".TrappeEntree_Ouvert := "IO_TrappeEntree_Ouvert";
	    
	    //___ %I2.5 - IO_TrappeEntree_Fermee
	    "St3_In".TrappeEntree_Fermee := "IO_TrappeEntree_Fermee";
	    
	    //___ %I2.6 - Trappe de sortie : Ouverte
	    "St3_In".TrappeSortie_Ouvert := "IO_TrappeSortie_Ouvert";
	    
	    //___ %I2.7 - Trappe de sortie : Fermée
	    "St3_In".TrappeSortie_Fermee := "IO_TrappeSortie_Fermee";
	    
	    //___ %I3.0 - Obturateur : Ouvert
	    "St3_In".Obturateur_Ouvert := "IO_Obturateur_Ouvert";
	    
	    //___ %I3.1 - Obturateur : Fermé
	    "St3_In".Obturateur_Fermee := "IO_Obturateur_Fermee";
	    
	    //___ %I3.2 - Porte RX : Ouverte (Homme)
	    "St3_In".PorteRX_Ouvert := "IO_PorteRX_Ouvert";
	    
	    //___ %I3.3 - Porte RX : Ferméee (Homme)
	    "St3_In".PorteRX_Fermee := "IO_PorteRX_Fermee";
	    
	    //___ %I3.4 - Présence barquette en début de RX : RX1
	    "St3_In".Cpt_RX1 := "IO_Cpt_RX1";
	    
	    //___ %I3.5 - Détection butée à came : RX2
	    "St3_In".Cpt_RX2 := "IO_Cpt_RX2";
	    
	    //___ %I3.6 - Détection butée pivot : RX3
	    "St3_In".Cpt_RX3 := "IO_Cpt_RX3";
	    
	    //___ %I3.7 - Obturateur Fermée + RX Actif
	    "St3_In".Vy_Orange := "IO_Vy_Orange";
	    
	    //___ %I4.0 - Obturateur Ouvert + RX Actif
	    "St3_In".Vy_Rouge := "IO_Vy_Rouge";
	    
	
	                   (* Output *)
	    
	    //___ %Q1.6 - Ouverture : Trappe d'entrée
	    "IO_Ouverture_TrappeEntree" := "St3_Out".Ouverture_TrappeEntree;
	    
	    //___ %Q1.7 - Fermeture : Trappe de sortie
	    "IO_Fermeture_TrappeEntree" := "St3_Out".Fermeture_TrappeEntree;
	    
	    //___ %Q2.0 - Ouverture : Trappe de sortie
	    "IO_Ouverture_TrappeSortie" := "St3_Out".Ouverture_TrappeSortie;
	    
	    //___ %Q2.1 - Fermeture : Trappe de sortie
	    "IO_Fermeture_TrappeSortie" := "St3_Out".Fermeture_TrappeSortie;
	    
	    //___ %Q2.3 - Ouverture : Obturateur
	    "IO_Ouverture_Obturateur" := "St3_Out".Ouverture_Obturateur;
	    
	    //___ %Q2.4 - Fermeture : Obturateur
	    "IO_Fermeture_Obturateur" := "St3_Out".Fermeture_Obturateur;
	    
	    //___ %Q2.5 - Ouverte : Porte RX (Homme)
	    "IO_Femerture_PorteRX" := "St3_Out".Femerture_PorteRX;
	    
	    //___ %Q2.6 - Fermeture : Porte RX (Homme)
	    "IO_Ouverture_PorteRX" := "St3_Out".Ouverture_PorteRX;
	    
	    
	    
END_FUNCTION

FUNCTION "IO_St4" : Void
{ S7_Optimized_Access := 'TRUE' }
VERSION : 0.1

BEGIN
	
	        (* IO - Station 4 : Dechargement  *)
	
	
	                  (* Input *)
	
	    //___ %I4.1 - Loquet haut : Pas de déplacement barquette 
	    "St4_In".Loquet_Haut := "IO_Loquet_Haut";
	    
	    //___ %I4.2 - Présence pile en zone de marquage
	    "St4_In".Cpt_M := "IO_Cpt_M";
	    
	    //___ %I4.3 - Pinces de préhension Déchagement C : Ouverte
	    "St4_In".PincesDC_Ouvert := "IO_PincesDC_Ouvert";
	    
	    //___ %I4.4 - Pinces de préhension Déchagement  C : Fermée
	    "St4_In".PincesDC_Fermee := "IO_PincesDC_Fermee";
	    
	    //___ %I4.5 - Présence pile en zone Déchagement C1
	    "St4_In".Cpt_DC1 := "IO_Cpt_DC1";
	    
	    //___ %I4.6 - Présence pile en zone Déchagement : C2
	    "St4_In".Cpt_DC2 := "IO_Cpt_DC2";
	    
	    //___ %I4.7 - Poussoir C en position : Haut
	    "St4_In".PoussoirC_Haut := "IO_PoussoirC_Haut";
	    
	    //___ %5.0 - Pinces de préhension Déchagement  NC : Ouverte
	    "St4_In".PincesDNC_Ouvert := "IO_PincesDNC_Ouvert";
	    
	    //___ %5.1 - Pinces de préhension Déchagement NC : Ferméee
	    "St4_In".PincesDNC_Fermee := "IO_PincesDNC_Fermee";
	    
	    //___ %5.2 - Présence pile en zone Déchagement NC0
	    "St4_In".Cpt_DNC0 := "IO_Cpt_DNC0";
	    
	    //___ %5.3 - Présence pile en zone Déchagement  DNC1
	    "St4_In".Cpt_DNC1 := "IO_Cpt_DNC1";
	    
	    //___ %5.4 - Présence pile en zone Déchagement DNC2
	    "St4_In".Cpt_DNC2 := "IO_Cpt_DNC2";
	    
	    //___ %5.5 - Poussoir NC en position : Haut
	    "St4_In".PoussoirNC_Haut := "IO_PoussoirNC_Haut";
	    
	    
	                   (* Output *)
	    
	    //___ %Q2.6 - Sortir : Loquet (Déplacement Barquette)
	    "IO_Sortir_Loquet" := "St4_Out".Sortir_Loquet;
	    
	    //___ %Q2.7 - Sortir : Poussoir Z-OK
	    "IO_Sortir_PoussoirC" := "St4_Out".Sortir_PoussoirC;
	    
	    //___ %Q3.0 - Ouverture : Pinces C
	    "IO_Ouverture_PincesC" := "St4_Out".Ouverture_PincesC;
	    
	    //___ %Q3.1 - Fermeture : Pinces C
	    "IO_Fermeture_PincesC":= "St4_Out".Fermeture_PincesC;
	    
	    //___ %Q3.2 - Zone Conforme pleine - A vidanger
	    "IO_Vy_C" := "St4_Out".Vy_C;
	    
	    //___ %Q3.3 - Sortir Poussoir NC
	    "IO_Sortir_PoussoirNC" := "St4_Out".Sortir_PoussoirNC;
	    
	    //___ %Q3.4 - Ouverture Pinces NC
	    "IO_Ouverture_PincesNC":= "St4_Out".Ouverture_PincesNC;
	    
	    //___ %Q3.5 - Fermeture Pinces NC
	    "IO_Fermeture_PincesNC" := "St4_Out".Ouverture_PincesNC;
	    
	    //___ %Q3.6 - Zone Non-Conforme pleine - A vidanger
	    "IO_Vy_NC" := "St4_Out".Vy_NC;
	    
	    
	    
	    
	    
END_FUNCTION

FUNCTION "G7A_St1" : Void   // FC110, LAD
{ S7_Optimized_Access := 'TRUE' }
VERSION : 0.1
// stored: AutoNumber false, IsIECCheckEnabled false, SetENOAutomatically false, UDAEnableTagReadback false
BEGIN

REGION Network 1: G7 Auto --> Station 1 : Empilement
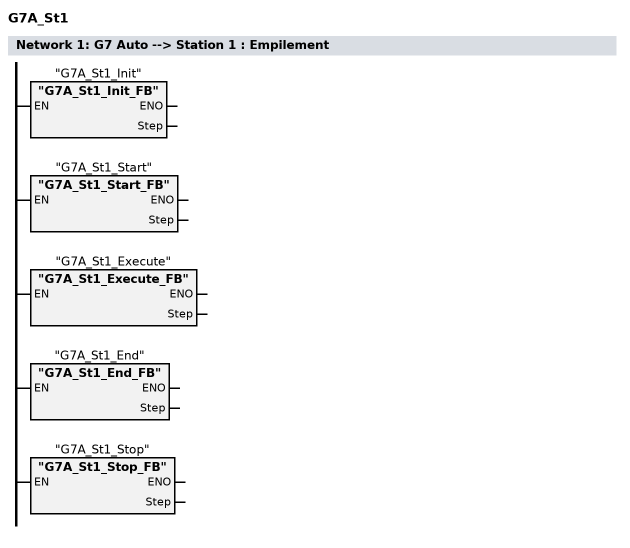
   RUNG wire#powerrail
      "G7A_St1_Init"("Step" =>)
   END_RUNG
   RUNG wire#powerrail
      "G7A_St1_Start"("Step" =>)
   END_RUNG
   RUNG wire#powerrail
      "G7A_St1_Execute"("Step" =>)
   END_RUNG
   RUNG wire#powerrail
      "G7A_St1_End"("Step" =>)
   END_RUNG
   RUNG wire#powerrail
      "G7A_St1_Stop"("Step" =>)
   END_RUNG
   // the same network as SCL:
   "G7A_St1_Init"();   // "G7A_St1_Init_FB"
   "G7A_St1_Start"();   // "G7A_St1_Start_FB"
   "G7A_St1_Execute"();   // "G7A_St1_Execute_FB"
   "G7A_St1_End"();   // "G7A_St1_End_FB"
   "G7A_St1_Stop"();   // "G7A_St1_Stop_FB"
END_REGION
END_FUNCTION

FUNCTION_BLOCK "G7A_St1_Init_FB"
{ S7_Optimized_Access := 'TRUE' }
VERSION : 0.1
   VAR_OUTPUT 
      Step : Int;
   END_VAR

   VAR 
      Step_100 { ExternalAccessible := 'False'; ExternalVisible := 'False'; ExternalWritable := 'False'} : Int;
      Authorization { ExternalAccessible := 'False'; ExternalVisible := 'False'; ExternalWritable := 'False'} : Bool;
   END_VAR


BEGIN
	                
	                (* G7 Auto : Init
	               Station 1 : Dépilement *)
	
	// Etape en cours
	    #Step := #Step_100;
	
	CASE #Step_100 OF
	        
	    0:  // Etape Init
	        #Step_100 := 10;
	        
	END_CASE;
	
	
	
END_FUNCTION_BLOCK

FUNCTION_BLOCK "G7A_St1_Start_FB"
{ S7_Optimized_Access := 'TRUE' }
VERSION : 0.1
   VAR_OUTPUT 
      Step : Int;
   END_VAR

   VAR 
      Step_100 { ExternalAccessible := 'False'; ExternalVisible := 'False'; ExternalWritable := 'False'} : Int;
      Authorization : Bool;
   END_VAR


BEGIN
	                
	                (* G7 Auto : Start
	               Station 1 : Dépilement *)
	
	// Etape en cours
	    #Step := #Step_100;
	
	CASE #Step_100 OF
	        
	    0:  // Etape Init
	        #Step_100 := 10;
	        
	END_CASE;
	
END_FUNCTION_BLOCK

FUNCTION_BLOCK "G7A_St1_Execute_FB"
{ S7_Optimized_Access := 'TRUE' }
VERSION : 0.1
   VAR_OUTPUT 
      Step : Int;
   END_VAR

   VAR 
      Step_100 { ExternalAccessible := 'False'; ExternalVisible := 'False'; ExternalWritable := 'False'} : Int;
      Authorization : Bool;
   END_VAR


BEGIN
	                
	                (* G7 Auto : Execute
	               Station 1 : Dépilement *)
	
	// Etape en cours
	    #Step := #Step_100;
	
	CASE #Step_100 OF
	        
	    0:  // Etape Init
	        #Step_100 := 10;
	        
	END_CASE;
END_FUNCTION_BLOCK

FUNCTION_BLOCK "G7A_St1_End_FB"
{ S7_Optimized_Access := 'TRUE' }
VERSION : 0.1
   VAR_OUTPUT 
      Step : Int;
   END_VAR

   VAR 
      Step_100 { ExternalAccessible := 'False'; ExternalVisible := 'False'; ExternalWritable := 'False'} : Int;
      Authorization : Bool;
   END_VAR


BEGIN
	                
	                 (* G7 Auto : End
	               Station 1 : Dépilement *)
	
	// Etape en cours
	    #Step := #Step_100;
	
	CASE #Step_100 OF
	        
	    0:  // Etape Init
	        #Step_100 := 10;
	        
	END_CASE;
END_FUNCTION_BLOCK

FUNCTION_BLOCK "G7A_St1_Stop_FB"
{ S7_Optimized_Access := 'TRUE' }
VERSION : 0.1
   VAR_OUTPUT 
      Step : Int;
   END_VAR

   VAR 
      Step_100 { ExternalAccessible := 'False'; ExternalVisible := 'False'; ExternalWritable := 'False'} : Int;
      Authorization : Bool;
   END_VAR


BEGIN
	                
	                (* G7 Auto : Stop
	               Station 1 : Dépilement *)
	
	// Etape en cours
	    #Step := #Step_100;
	
	CASE #Step_100 OF
	        
	    0:  // Etape Init
	        #Step_100 := 10;
	        
	END_CASE;
	
	
END_FUNCTION_BLOCK

FUNCTION "G7A_St2" : Void   // FC210, LAD
{ S7_Optimized_Access := 'TRUE' }
VERSION : 0.1
// stored: AutoNumber false, IsIECCheckEnabled false, SetENOAutomatically false, UDAEnableTagReadback false
BEGIN

REGION Network 1: G7 Auto --> Station 2 : Vision
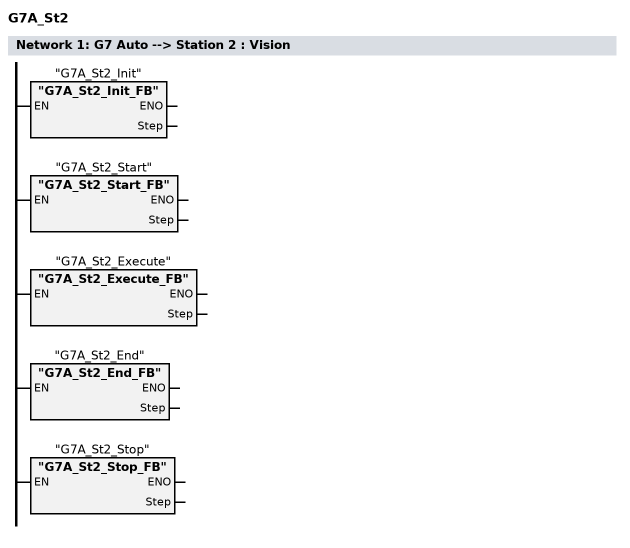
   RUNG wire#powerrail
      "G7A_St2_Init"("Step" =>)
   END_RUNG
   RUNG wire#powerrail
      "G7A_St2_Start"("Step" =>)
   END_RUNG
   RUNG wire#powerrail
      "G7A_St2_Execute"("Step" =>)
   END_RUNG
   RUNG wire#powerrail
      "G7A_St2_End"("Step" =>)
   END_RUNG
   RUNG wire#powerrail
      "G7A_St2_Stop"("Step" =>)
   END_RUNG
   // the same network as SCL:
   "G7A_St2_Init"();   // "G7A_St2_Init_FB"
   "G7A_St2_Start"();   // "G7A_St2_Start_FB"
   "G7A_St2_Execute"();   // "G7A_St2_Execute_FB"
   "G7A_St2_End"();   // "G7A_St2_End_FB"
   "G7A_St2_Stop"();   // "G7A_St2_Stop_FB"
END_REGION
END_FUNCTION

FUNCTION_BLOCK "G7A_St2_Init_FB"
{ S7_Optimized_Access := 'TRUE' }
VERSION : 0.1
   VAR_OUTPUT 
      Step : Int;
   END_VAR

   VAR 
      Step_100 { ExternalAccessible := 'False'; ExternalVisible := 'False'; ExternalWritable := 'False'} : Int;
      Authorization : Bool;
   END_VAR


BEGIN
	                
	                (* G7 Auto : Init
	               Station 2 : Vision *)
	
	// Etape en cours
	    #Step := #Step_100;
	
	CASE #Step_100 OF
	        
	    0:  // Etape Init
	        #Step_100 := 10;
	        
	END_CASE;
END_FUNCTION_BLOCK

FUNCTION_BLOCK "G7A_St2_Start_FB"
{ S7_Optimized_Access := 'TRUE' }
VERSION : 0.1
   VAR_OUTPUT 
      Step : Int;
   END_VAR

   VAR 
      Step_100 { ExternalAccessible := 'False'; ExternalVisible := 'False'; ExternalWritable := 'False'} : Int;
      Authorization : Bool;
   END_VAR


BEGIN
	                
	                (* G7 Auto : Start
	                Station 2 : Vision *)
	
	// Etape en cours
	    #Step := #Step_100;
	
	CASE #Step_100 OF
	        
	    0:  // Etape Init
	        #Step_100 := 10;
	        
	END_CASE;
END_FUNCTION_BLOCK

FUNCTION_BLOCK "G7A_St2_Execute_FB"
{ S7_Optimized_Access := 'TRUE' }
VERSION : 0.1
   VAR_OUTPUT 
      Step : Int;
   END_VAR

   VAR 
      Step_100 { ExternalAccessible := 'False'; ExternalVisible := 'False'; ExternalWritable := 'False'} : Int;
      Authorization : Bool;
   END_VAR


BEGIN
	                
	                (* G7 Auto : Execute
	                 Station 2 : Vision *)
	
	// Etape en cours
	    #Step := #Step_100;
	
	CASE #Step_100 OF
	        
	    0:  // Etape Init
	        #Step_100 := 10;
	        
	END_CASE;
END_FUNCTION_BLOCK

FUNCTION_BLOCK "G7A_St2_End_FB"
{ S7_Optimized_Access := 'TRUE' }
VERSION : 0.1
   VAR_OUTPUT 
      Step : Int;
   END_VAR

   VAR 
      Step_100 { ExternalAccessible := 'False'; ExternalVisible := 'False'; ExternalWritable := 'False'} : Int;
      Authorization : Bool;
   END_VAR


BEGIN
	                
	                (* G7 Auto : End
	                Station 2 : Vision *)
	
	// Etape en cours
	    #Step := #Step_100;
	
	CASE #Step_100 OF
	        
	    0:  // Etape Init
	        #Step_100 := 10;
	        
	END_CASE;
END_FUNCTION_BLOCK

FUNCTION_BLOCK "G7A_St2_Stop_FB"
{ S7_Optimized_Access := 'TRUE' }
VERSION : 0.1
   VAR_OUTPUT 
      Step : Int;
   END_VAR

   VAR 
      Step_100 { ExternalAccessible := 'False'; ExternalVisible := 'False'; ExternalWritable := 'False'} : Int;
      Authorization : Bool;
   END_VAR


BEGIN
	                
	                (* G7 Auto : Stop
	                Station 2 : Vision *)
	
	// Etape en cours
	    #Step := #Step_100;
	
	CASE #Step_100 OF
	        
	    0:  // Etape Init
	        #Step_100 := 10;
	        
	END_CASE;
END_FUNCTION_BLOCK

FUNCTION "G7A_St3" : Void   // FC310, LAD
{ S7_Optimized_Access := 'TRUE' }
VERSION : 0.1
// stored: AutoNumber false, IsIECCheckEnabled false, SetENOAutomatically false, UDAEnableTagReadback false
BEGIN

REGION Network 1: G7 Auto --> Station 3 : RX
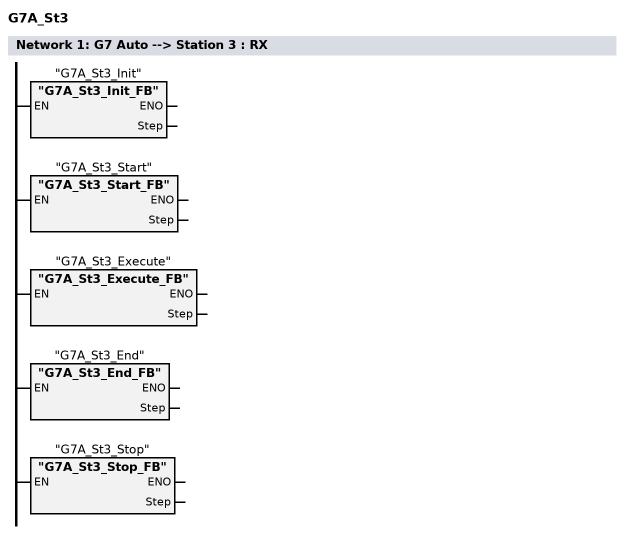
   RUNG wire#powerrail
      "G7A_St3_Init"("Step" =>)
   END_RUNG
   RUNG wire#powerrail
      "G7A_St3_Start"("Step" =>)
   END_RUNG
   RUNG wire#powerrail
      "G7A_St3_Execute"("Step" =>)
   END_RUNG
   RUNG wire#powerrail
      "G7A_St3_End"("Step" =>)
   END_RUNG
   RUNG wire#powerrail
      "G7A_St3_Stop"("Step" =>)
   END_RUNG
   // the same network as SCL:
   "G7A_St3_Init"();   // "G7A_St3_Init_FB"
   "G7A_St3_Start"();   // "G7A_St3_Start_FB"
   "G7A_St3_Execute"();   // "G7A_St3_Execute_FB"
   "G7A_St3_End"();   // "G7A_St3_End_FB"
   "G7A_St3_Stop"();   // "G7A_St3_Stop_FB"
END_REGION
END_FUNCTION

FUNCTION_BLOCK "G7A_St3_Init_FB"
{ S7_Optimized_Access := 'TRUE' }
VERSION : 0.1
   VAR_OUTPUT 
      Step : Int;
   END_VAR

   VAR 
      Step_100 { ExternalAccessible := 'False'; ExternalVisible := 'False'; ExternalWritable := 'False'} : Int;
      Authorization : Bool;
   END_VAR


BEGIN
	                
	                (* G7 Auto : Init
	                  Station 3 : RX *)
	
	// Etape en cours
	    #Step := #Step_100;
	
	CASE #Step_100 OF
	        
	    0:  // Etape Init
	        #Step_100 := 10;
	        
	END_CASE;
	
	
	
END_FUNCTION_BLOCK

FUNCTION_BLOCK "G7A_St3_Start_FB"
{ S7_Optimized_Access := 'TRUE' }
VERSION : 0.1
   VAR_OUTPUT 
      Step : Int;
   END_VAR

   VAR 
      Step_100 { ExternalAccessible := 'False'; ExternalVisible := 'False'; ExternalWritable := 'False'} : Int;
      Authorization : Bool;
   END_VAR


BEGIN
	                
	                (* G7 Auto : Start
	                  Station 3 : RX *)
	
	// Etape en cours
	    #Step := #Step_100;
	
	CASE #Step_100 OF
	        
	    0:  // Etape Init
	        #Step_100 := 10;
	        
	END_CASE;
END_FUNCTION_BLOCK

FUNCTION_BLOCK "G7A_St3_Execute_FB"
{ S7_Optimized_Access := 'TRUE' }
VERSION : 0.1
   VAR_OUTPUT 
      Step : Int;
   END_VAR

   VAR 
      Step_100 { ExternalAccessible := 'False'; ExternalVisible := 'False'; ExternalWritable := 'False'} : Int;
      Authorization : Bool;
   END_VAR


BEGIN
	                
	                (* G7 Auto : Execute
	                   Station 3 : RX *)
	
	// Etape en cours
	    #Step := #Step_100;
	
	CASE #Step_100 OF
	        
	    0:  // Etape Init
	        #Step_100 := 10;
	        
	END_CASE;
END_FUNCTION_BLOCK

FUNCTION_BLOCK "G7A_St3_End_FB"
{ S7_Optimized_Access := 'TRUE' }
VERSION : 0.1
   VAR_OUTPUT 
      Step : Int;
   END_VAR

   VAR 
      Step_100 { ExternalAccessible := 'False'; ExternalVisible := 'False'; ExternalWritable := 'False'} : Int;
      Authorization : Bool;
   END_VAR


BEGIN
	                
	                (* G7 Auto : End
	                  Station 3 : RX *)
	
	// Etape en cours
	    #Step := #Step_100;
	
	CASE #Step_100 OF
	        
	    0:  // Etape Init
	        #Step_100 := 10;
	        
	END_CASE;
END_FUNCTION_BLOCK

FUNCTION_BLOCK "G7A_St3_Stop_FB"
{ S7_Optimized_Access := 'TRUE' }
VERSION : 0.1
   VAR_OUTPUT 
      Step : Int;
   END_VAR

   VAR 
      Step_100 { ExternalAccessible := 'False'; ExternalVisible := 'False'; ExternalWritable := 'False'} : Int;
      Authorization : Bool;
   END_VAR


BEGIN
	                
	                (* G7 Auto : Stop
	                  Station 3 : RX *)
	
	// Etape en cours
	    #Step := #Step_100;
	
	CASE #Step_100 OF
	        
	    0:  // Etape Init
	        #Step_100 := 10;
	        
	END_CASE;
END_FUNCTION_BLOCK

FUNCTION "G7A_St4" : Void   // FC410, LAD
{ S7_Optimized_Access := 'TRUE' }
VERSION : 0.1
// stored: AutoNumber false, IsIECCheckEnabled false, SetENOAutomatically false, UDAEnableTagReadback false
BEGIN

REGION Network 1: G7 Auto --> Station 4 : Marquage
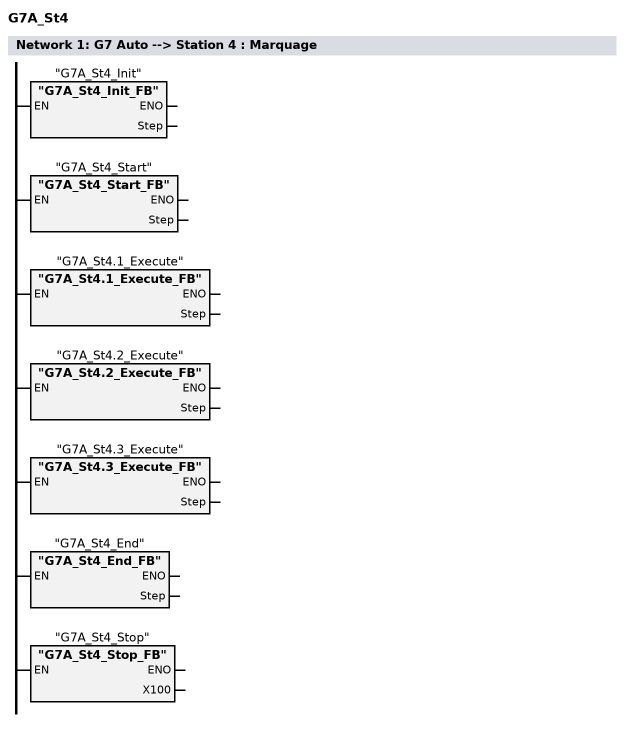
   RUNG wire#powerrail
      "G7A_St4_Init"("Step" =>)
   END_RUNG
   RUNG wire#powerrail
      "G7A_St4_Start"("Step" =>)
   END_RUNG
   RUNG wire#powerrail
      "G7A_St4.1_Execute"("Step" =>)
   END_RUNG
   RUNG wire#powerrail
      "G7A_St4.2_Execute"("Step" =>)
   END_RUNG
   RUNG wire#powerrail
      "G7A_St4.3_Execute"("Step" =>)
   END_RUNG
   RUNG wire#powerrail
      "G7A_St4_End"("Step" =>)
   END_RUNG
   RUNG wire#powerrail
      "G7A_St4_Stop"(X100 =>)
   END_RUNG
   // the same network as SCL:
   "G7A_St4_Init"();   // "G7A_St4_Init_FB"
   "G7A_St4_Start"();   // "G7A_St4_Start_FB"
   "G7A_St4.1_Execute"();   // "G7A_St4.1_Execute_FB"
   "G7A_St4.2_Execute"();   // "G7A_St4.2_Execute_FB"
   "G7A_St4.3_Execute"();   // "G7A_St4.3_Execute_FB"
   "G7A_St4_End"();   // "G7A_St4_End_FB"
   "G7A_St4_Stop"();   // "G7A_St4_Stop_FB"
END_REGION
END_FUNCTION

FUNCTION_BLOCK "G7A_St4_Init_FB"
{ S7_Optimized_Access := 'TRUE' }
VERSION : 0.1
   VAR_OUTPUT 
      Step : Int;
   END_VAR

   VAR 
      Step_100 { ExternalAccessible := 'False'; ExternalVisible := 'False'; ExternalWritable := 'False'} : Int;
      Authorization : Bool;
   END_VAR


BEGIN
	                
	                (* G7 Auto : Init
	            Station 4 : Déchargement *)
	
	// Etape en cours
	    #Step := #Step_100;
	    
	CASE #Step_100 OF
	        
	    0:  // Etape Init
	        #Step_100 := 10;
	        
	END_CASE;
END_FUNCTION_BLOCK

FUNCTION_BLOCK "G7A_St4_Start_FB"
{ S7_Optimized_Access := 'TRUE' }
VERSION : 0.1
   VAR_OUTPUT 
      Step : Int;
   END_VAR

   VAR 
      Step_100 { ExternalAccessible := 'False'; ExternalVisible := 'False'; ExternalWritable := 'False'} : Int;
      Authorization : Bool;
   END_VAR


BEGIN
	                
	                (* G7 Auto : Start
	            Station 4 : Déchargement *)
	
	// Etape en cours
	    #Step := #Step_100;
	    
	CASE #Step_100 OF
	        
	    0:  // Etape Init
	        #Step_100 := 10;
	        
	END_CASE;
END_FUNCTION_BLOCK

FUNCTION_BLOCK "G7A_St4.1_Execute_FB"
{ S7_Optimized_Access := 'TRUE' }
VERSION : 0.1
   VAR_OUTPUT 
      Step : Int;
   END_VAR

   VAR 
      Step_100 { ExternalAccessible := 'False'; ExternalVisible := 'False'; ExternalWritable := 'False'} : Int;
      Authorization : Bool;
   END_VAR


BEGIN
	                
	                (* G7 Auto : Execute
	                Station 4 : Marquage *)
	
	// Etape en cours
	    #Step := #Step_100;
	
	CASE #Step_100 OF
	        
	    0:  // Etape Init
	        #Step_100 := 10;
	        
	END_CASE;
END_FUNCTION_BLOCK

FUNCTION_BLOCK "G7A_St4.2_Execute_FB"
{ S7_Optimized_Access := 'TRUE' }
VERSION : 0.1
   VAR_OUTPUT 
      Step : Int;
   END_VAR

   VAR 
      Step_100 : Int;
   END_VAR


BEGIN
	                
	                      (* G7 Auto : Start
	               Station 4 : Empilement Conforme *)
	
	// Etape en cours
	#Step := #Step_100;
	
	CASE #Step_100 OF
	        
	    0:  // Etape Init
	        #Step_100 := 10;
	        
	END_CASE;
END_FUNCTION_BLOCK

FUNCTION_BLOCK "G7A_St4.3_Execute_FB"
{ S7_Optimized_Access := 'TRUE' }
VERSION : 0.1
   VAR_OUTPUT 
      Step : Int;
   END_VAR

   VAR 
      Step_100 : Int;
   END_VAR


BEGIN
	                
	                      (* G7 Auto : Start
	               Station 4 : Empilement Non-Conforme *)
	
	// Etape en cours
	#Step := #Step_100;
	
	CASE #Step_100 OF
	        
	    0:  // Etape Init
	        #Step_100 := 10;
	        
	END_CASE;
END_FUNCTION_BLOCK

FUNCTION_BLOCK "G7A_St4_End_FB"
{ S7_Optimized_Access := 'TRUE' }
VERSION : 0.1
   VAR_OUTPUT 
      Step : Int;
   END_VAR

   VAR 
      Step_100 { ExternalAccessible := 'False'; ExternalVisible := 'False'; ExternalWritable := 'False'} : Int;
      Authorization : Bool;
   END_VAR


BEGIN
	                
	                (* G7 Auto : End
	            Station 4 : Déchargement *)
	
	// Etape en cours
	    #Step := #Step_100;
	    
	CASE #Step_100 OF
	        
	    0:  // Etape Init
	        #Step_100 := 10;
	        
	END_CASE;
END_FUNCTION_BLOCK

FUNCTION_BLOCK "G7A_St4_Stop_FB"
{ S7_Optimized_Access := 'TRUE' }
VERSION : 0.1
   VAR_OUTPUT 
      X100 : Int;
   END_VAR

   VAR 
      Step_100 { ExternalAccessible := 'False'; ExternalVisible := 'False'; ExternalWritable := 'False'} : Int;
      Authorization : Bool;
   END_VAR


BEGIN
	                
	                (* G7 Auto : Stop
	            Station 4 : Déchargement *)
	
	// Etape en cours
	    #X100 := #Step_100;
	
	CASE #Step_100 OF
	        
	    0:  // Etape Init
	        #Step_100 := 10;
	        
	END_CASE;
	
	
END_FUNCTION_BLOCK

FUNCTION_BLOCK "Obj_St1_FB"   // FB100, FBD
{ S7_Optimized_Access := 'TRUE' }
VERSION : 0.1
// stored: AutoNumber false, IsIECCheckEnabled false, IsRetainMemResEnabled false, MemoryReserve 100, SetENOAutomatically false, UDAEnableTagReadback false
   VAR
      Axe_X : Struct
         _ActPos : Real;
         _ActVel : Real;
         _Mode : Int;
         Home : Bool;
         Halt : Bool;
         Jog : Bool;
         MoveAbs : Bool;
         MoveRel : Bool;
         MoveVel : Bool;
         PowerOff : Bool;
         PowerOn : Bool;
         SensPos : Bool;
         SensNeg : Bool;
         xBusy : Bool;
         xHomed : Bool;
         xMoveAbsDone : Bool;
         xMoveRelDone : Bool;
         xPower : Bool;
      END_STRUCT;
      Axe_Y : Struct
         _ActPos : Real;
         _ActVel : Real;
         _Mode : Int;
         Home : Bool;
         Halt : Bool;
         Jog : Bool;
         MoveAbs : Bool;
         MoveRel : Bool;
         MoveVel : Bool;
         PowerOff : Bool;
         PowerOn : Bool;
         SensPos : Bool;
         SensNeg : Bool;
         xBusy : Bool;
         xHomed : Bool;
         xMoveAbsDone : Bool;
         xMoveRelDone : Bool;
         xPower : Bool;
      END_STRUCT;
      Prehenseur_Z : Struct
         _ActPos : Real;
         _ActVel : Real;
         _Mode : Int;
         Home : Bool;
         Halt : Bool;
         Jog : Bool;
         MoveAbs : Bool;
         MoveRel : Bool;
         MoveVel : Bool;
         PowerOff : Bool;
         PowerOn : Bool;
         SensPos : Bool;
         SensNeg : Bool;
         xBusy : Bool;
         xHomed : Bool;
         xMoveAbsDone : Bool;
         xMoveRelDone : Bool;
         xPower : Bool;
      END_STRUCT;
   END_VAR
BEGIN

REGION Network 1: Station 1 - Axe X
   // //___ ModePose : 
   //          1 ---> Relative positioning
   //          2 ---> Absolute positioning
   //          3 ---> Not supported
   //          4 ---> Referencing - referencing point approach
   //          5 ---> Referencing - set referencing point
   //          6 ---> Traversing block (record mode)
   //          7 ---> Jog
   //          8 ---> Not supported
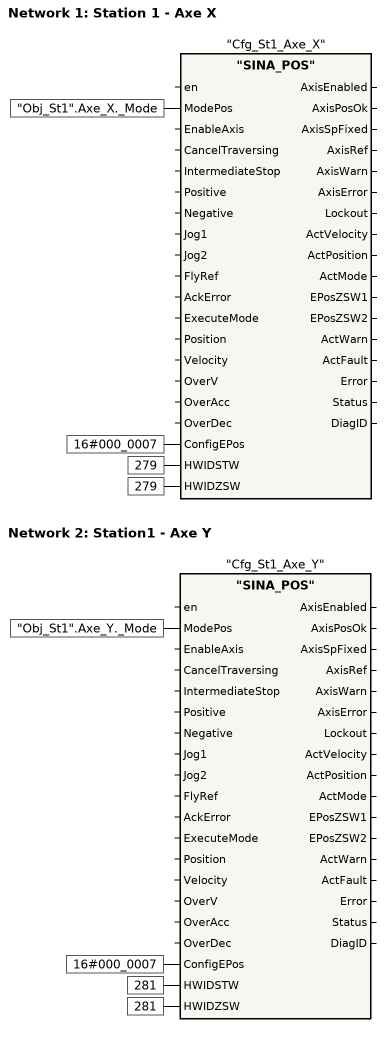
   "Cfg_St1_Axe_X"(ModePos := "Obj_St1".Axe_X._Mode, ConfigEPos := 16#000_0007, HWIDSTW := 279, HWIDZSW := 279);   // "SINA_POS"
END_REGION

REGION Network 2: Station1 - Axe Y
   // //___ ModePose : 
   //          1 ---> Relative positioning
   //          2 ---> Absolute positioning
   //          3 ---> Not supported
   //          4 ---> Referencing - referencing point approach
   //          5 ---> Referencing - set referencing point
   //          6 ---> Traversing block (record mode)
   //          7 ---> Jog
   //          8 ---> Not supported
   "Cfg_St1_Axe_Y"(ModePos := "Obj_St1".Axe_Y._Mode, ConfigEPos := 16#000_0007, HWIDSTW := 281, HWIDZSW := 281);   // "SINA_POS"
END_REGION

REGION Network 3: Station 1 - Prehenseur Z
   // //___ ModePose : 
   //          1 ---> Relative positioning
   //          2 ---> Absolute positioning
   //          3 ---> Not supported
   //          4 ---> Referencing - referencing point approach
   //          5 ---> Referencing - set referencing point
   //          6 ---> Traversing block (record mode)
   //          7 ---> Jog
   //          8 ---> Not supported
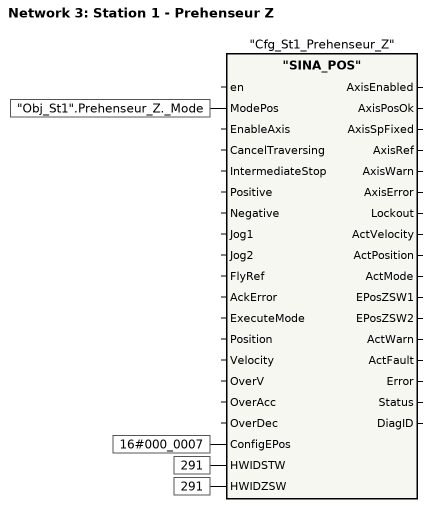
   "Cfg_St1_Prehenseur_Z"(ModePos := "Obj_St1".Prehenseur_Z._Mode,   // "SINA_POS"
                          ConfigEPos := 16#000_0007,
                          HWIDSTW := 291,
                          HWIDZSW := 291);
END_REGION
END_FUNCTION_BLOCK

FUNCTION_BLOCK "SINA_POS"
TITLE = 'Positioning with SINAMICS and S7'
{ S7_Optimized_Access := 'TRUE' }
AUTHOR : DRVDPS7
FAMILY : DRIVES
NAME : SINA_POS
VERSION : 5.7
//Copyright (C) Siemens AG 2012. All Rights Reserved. Confidential
//-------------------------------------------------------------------------------------- 
//SINA_POS: Positionierung mit dem Antriebsbaustein SINAMICS S120/G120 <-> S7-1200
//------------------------------------------------------------------------------------- Ersteller: Siemens AG Erlangen A&D MC PM   Datum:  07.07.10        Vers.:2.1
//Änderung:  J.B. Typical Team                       18.12.12              2.2
//    Umsetzung in SCL / TIA 
//Änderung:  J.B. Typical Team                       18.04.13              2.3
//    Bei Betriebsart "Referenzieren - Referenzpunkt setzen"
//    nicht intern setzen sondern Eingang #Execute abfragen als 
//    Startbedingung
//Änderung:  J.B. Typical Team                       29.04.13              2.4
//    1. Off1 möglich bei ungültige Betriebsart
//    2. Referenzpunkt setzen Exceute übernehmen
//    3. Fehlermeldung ausgeben bei Wechel ohne 
//       Beendigung der Betriebsart 
//    4. "Q" an den Ausgänge entfernen
//    5. Neuer Ausgang PwrInhibit
//     
//Änderung:  J.B. Typical Team                       14.05.13              2.5
//    Fehlerbehebung und Defaultwerte ändern
//Änderung:  J.B. Typical Team                       28.06.13              2.6
//    HW-Zugriffsermittlung über LOG2MOD
//Änderung:  J.B. Typical Team                       18.07.13              2.7
//    HW-Zugriffsermittlung über zwei HW-Eingänge
//Änderung:  J.B. Typical Team                       18.09.13              2.8
//    Konvertierungsfehler behoben
//Änderung:  J.B. Typical Team                       25.09.13              2.9
//    Bei Betriebswechsel von 3 nach 6 darf MidStart nicht sitzen
//Änderung:  J.B. Typical Team                       31.03.14              3.0
//    In der Betriebsart 1-3 und 6 darf MidTrTyp nicht sitzen
//Änderung:  J.B. Typical Team                       25.06.14              3.1
//    Das Quittierbit "AckFlt" immer durchreichen
//Änderung:  J.B. Typical Team                       30.07.14              4.0
//    Festlegung auf einheitlicher neuer Version 4.0
//Änderung:  J.B. Typical Team                       07.11.14              4.1
//    Fehlerbehebung falsche Zuweisung von Off1 bei Mode 4
//    und Mode 8(DriveLib V4 - RQ 346046)
//Änderung:  F.G. Typical Team                       16.04.15              4.2
//    Anzahl der Zyklen die auf die Rückmeldung fliegendes Ref.
//    gewartet wird verdoppelt (siRetryMax = 10)  (DriveLib V4 - RQ 367986)
//Änderung:  F.G. Typical Team                       15.09.15              4.3
//    Anzahl der Zyklen die auf die Rückmeldung fliegendes Ref.
//    gewartet noch einmal um 5 erhöht (siRetryMax = 15)  (DriveLib V4 - RQ 367986)
//Änderung:  F.G. Typical Team                       15.09.15              4.4
//    Abfrage des richtigen Bits im EPosZSW1 (Zeile 1394)es muss das Bit12 
//    und nicht das Bit 11 abgefragt werden  (DriveLib V4 - RQ 367986)
//Änderung:  F.G. Typical Team                       03.12.15              4.5
//    1. Ein-/Ausgänge an Programmierleitfaden für TIA-Portal angepasst
//       Zusätzlicher Eingang um alle Bits in den STWs zu bedienen
//    2. Warnung durch Initialisierung elimininiert
//Änderung:  F.G. Typical Team                       13.09.16              4.6
//    Ausgabewerte am Ausgang "Status" angepasst 
//
//Änderung:  G.F. Typical Team                       11.01.17              5.0
//    - Festlegung auf einheitlicher neuer Version 5.0 
//
//Änderung:  G.F. Typical Team                       13.07.17              5.1
//    - Zuordnung der Bits von ConfigPos korrigiert 
//
//Änderung:  G.F. Typical Team                       12.01.18              5.2
//    - RQ2637983 sxSendBuf.EPosSTW2.%X1 in Mode 7 und 8 rücksetzen 
//Änderung:  G.F. Typical Team                       20.07.18              5.3
//    - ZSW1.13 als Ausgang zur Verfügung gestellt (wegen FW - Änderung)
//Änderung:  G.F. Typical Team                       18.10.18              5.4
//    - RQ 824321 Zähler für fliegendes Referenzieren zurücksetzen
//Änderung:  G.F. Typical Team                       08.02.19              5.5
//    - Version wegen Änderungen in älteren Lib-Versionen 
//Änderung:  G.F. Typical Team                       08.02.19              5.6
//    - RQ 3901129 Fehler Flankenauswertung Eingang ExecuteMode behoben Bibliothek V7
//Änderung:  G.F. Typical Team                       17.05.19              5.7
//    - RQ 4094299 Fehler Referenzfahrt wird nicht gestartet behoben Bibliothek V7
//Funktion: Positionierung mit dem Antriebsbaustein SINAMICS S120/G120 <-> S7-1200
//********************************************************************************************************************************************************
//************************************************************************FB283***************************************************************************
//********************************************************************************************************************************************************
   VAR_INPUT 
      ModePos : Int := 0;   // Settings of the mode
      EnableAxis : Bool := 0;   // 1 = Enable the drive
      CancelTraversing : Bool := 1;   // 0 = Reject active traverse task
      IntermediateStop : Bool := 1;   // 0 = Intermediate STOP of traverse command
      Positive : Bool := 0;   // 1 = Direction positive
      Negative : Bool := 0;   // 1 = Direction negative
      Jog1 : Bool := 0;   // 1 = Use jog 1 (direction / speed)
      Jog2 : Bool := 0;   // 1 = Use jog 2 (direction / speed)
      FlyRef : Bool := 0;   // 1 = Start flying reference function
      AckError : Bool := 0;   // 1  = Acknowledge of errors
      ExecuteMode : Bool := 0;   // 0-->1 = Start the mode
      Position : DInt := 0;   // Position of the MDI mode or setting of traversing block
      Velocity : DInt := 0;   // MDI velocity
      OverV : Int := 100;   // Override of  velocity in [%] --> 4000h=100%
      OverAcc : Int := 100;   // Override of acceleration in [%] --> 4000h=100%
      OverDec : Int := 100;   // Override of deceleration in [%] --> 4000h=100%
      ConfigEPos : DWord := 16#0000_0003;   // binary programmed input to control all functions in the telegram without its own function block input
      HWIDSTW : HW_IO := 0;   // Hardware Identifer set point slot
      HWIDZSW : HW_IO := 0;   // Hardware Identifer actual value slot
   END_VAR

   VAR_OUTPUT 
      AxisEnabled : Bool := 0;   // 1= Axis in operation
      AxisPosOk : Bool := 0;   // 1= Position setpoint reached
      AxisSpFixed : Bool := 0;   // 1= Setpoint fixed (Attention: Dependence on SINAMICS firmware)
      AxisRef : Bool := 0;   // 1= Reference point set
      AxisWarn : Bool := 0;   // 1= Axis alarm / warning present
      AxisError : Bool := 0;   // 1= Axis fault present
      Lockout : Bool := 0;   // 1= Axis in lockout state
      ActVelocity : DInt := 0;   // Actual drive speed (has to be normed with p2000 --> 40000000h = 100%)
      ActPosition : DInt := 0;   // Actual position in [LU]
      ActMode : Int := 0;   // Active EPos mode
      EPosZSW1 : Word := 0;   // Status of EPOS ZSW1
      EPosZSW2 : Word := 0;   // Status of EPOS ZSW2
      ActWarn : Word := 0;   // Actual number of warning
      ActFault : Word := 0;   // Actual number of error
      Error : Bool := 0;   // 1 = Error  (FB and Infeed)
      Status : Word := 0;   // Status output (7002 = FB in operation; 8xxx = error description  - read the manual)
      DiagID : Word := 0;   // Error codes of the cyclic system funtion blocks DPWR / DPRD_DAT
   END_VAR

   VAR 
      sbOff1Edge : Bool := 0;   // Positive edge of starting or stopping the device
      sbOff1 : Bool := 0;   // Starting or stopping the device
      sbExecuteEdge : Bool := 0;   // Positive edge of activate traversing block
      sbExecute : Bool := 0;   // Activate traversing block
      sbRefTypEdge : Bool := 0;   // Positive edge of referencing type "flying reference"
      sbRefTyp : Bool := 0;   // Referencing type "flying reference"
      sbMdiStart : Bool := 0;   // Direct setpoint input / MDI - start
      sbMdiStartEdge : Bool := 0;   // Positive edge of direct setpoint input / MDI - start
      sbRefStart : Bool := 0;   // Referencing start
      sbJogInc : Bool := 0;   // Jogging incremental
      sbReady : Bool := 0;   // Ready to power up / to start
      sbIOp : Bool := 0;   // Ready to operate
      sbAccel : Bool := 0;   // Axis accelerating
      sbDecel : Bool := 0;   // Axis decelerating
      sbAlarm : Bool := 0;   // Alarm / Warnung present
      sbFault : Bool := 0;   // Fault present
      sbFWD : Bool := 0;   // Axis drives forwards
      sbBWD : Bool := 0;   // Axis drives backwards
      sbBusy : Bool := 0;   // Mode of operation is explained
      swStatus : Word := 16#0000;   // Mode of operation disturbance
      swEPosZSW1 : Word := 16#0000;   // Status of EPOS ZSW1
      swEPosZSW2 : Word := 16#0000;   // Status of EPOS ZSW2
      siExecuteCyc : Int := 0;   // Counter of runcycle of active traversing block
      siRefTypCyc : Int := 0;   // Counter of runcycle of referencing type "flying reference"
      siJogIncCyc : Int := 0;   // Counter of runcycle of jogging incremental
      siMdiStartCyc : Int := 0;   // Counter of runcycle of direct setpoint input / MDI - start
      siRefActRetry : Int := 0;   // Counter of retry of reference point approach active
      siModePos : Int := 0;   // Setting of mode
      siModePosMax : Int := 8;   // Max. count of mode
      siCycWait : Int := 5;   // Counter of cycle of waiting
      siRetryMax : Int := 30;   // Max. count of cycles of retry
      sbModePos : Bool := 0;   // Mode of setting okay
      sxSendBuf : Struct   // send buffer of telegram for sending data to the drive
         STW1 : Word := WORD#16#0000;   // STW1sxSTW1     : STRUCT            Jog1            : BOOL:=0;              // ST-Wort-1 Bit 08 --> 1 = Jogging - signal source 1            Jog2            : BOOL:=0;              // ST-Wort-1 Bit 09 --> 1 = Jogging - signal source 2            LB              : BOOL:=1; // Allways   // ST-Wort-1 Bit 10 --> 1 = Life bit             RefStart        : BOOL:=0;              // ST-Wort-1 Bit 11 --> 1 = Referencing start / stop            Bit12           : BOOL:=0;              // ST-Wort-1 Bit 12 --> 1 = Reserve            Bit13           : BOOL:=0;              // ST-Wort-1 Bit 13 --> 1 = Externer Satzwechsel            Bit14           : BOOL:=0;              // ST-Wort-1 Bit 14 --> 1 = Reserve            Bit15           : BOOL:=0;              // ST-Wort-1 Bit 15 --> 1 = Reserve            Off1            : BOOL:=0;              // ST-Wort-1 Bit 00 --> 1 = OFF1/ON (flanks acceptance)            Off2            : BOOL:=1; // Allways   // ST-Wort-1 Bit 01 --> 1 = OFF2/ON (enable possible)            Off3            : BOOL:=1; // Allways   // ST-Wort-1 Bit 02 --> 1 = OFF3/ON (enable possible)            Enc             : BOOL:=1; // Allways   // ST-Wort-1 Bit 03 --> 1 = Enable controller            RejTrvTsk       : BOOL:=0;              // ST-Wort-1 Bit 04 --> 1 = Traversing block and MDI - reject task            IntMStop        : BOOL:=0;              // ST-Wort-1 Bit 05 --> 1 = Traversing block and MDI - intermediate - STOP            TrvStart        : BOOL:=0;              // ST-Wort-1 Bit 06 --> 1 = Traversing start - direct setpoint input / MDI - transfer edge            AckFault        : BOOL:=0;              // ST-Wort-1 Bit 07 --> 1 = Acknowledge fault         END_STRUCT;
         EPosSTW1 : Word := WORD#16#0000;   // EPOSSTW1sxEPosSTW1   : STRUCT            MdiTyp          : BOOL:=0;              // EPOS-Wort-1 Bit 08 --> 1 = Direct setpoint input / MDI - positioning type            MdiPos          : BOOL:=0;              // EPOS-Wort-1 BIT 09 --> 1 = Direct setpoint input / MDI - positive direction            MdiNeg          : BOOL:=0;              // EPOS-Wort-1 BIT 10 --> 1 = Direct setpoint input / MDI - negative direction            Bit11           : BOOL:=0;              // EPOS-Wort-1 BIT 11 --> 1 = Reserve            MdiTrTyp        : BOOL:=0;              // EPOS-Wort-1 BIT 12 --> 1 = Direct setpoint input / MDI - transfer type            Bit13           : BOOL:=0;              // EPOS-Wort-1 BIT 13 --> 1 = Reserve            MdiSetup        : BOOL:=0;              // EPOS-Wort-1 BIT 14 --> 1 = Direct setpoint input / MDI - setup selection            MdiStart        : BOOL:=0;              // EPOS-Wort-1 BIT 15 --> 1 = Direct setpoint input / MDI - start              TrvBit0         : BOOL:=0;              // EPOS-Wort-1 BIT 00 --> 1 = Traversing block - block selection bit 0            TrvBit1         : BOOL:=0;              // EPOS-Wort-1 BIT 01 --> 1 = Traversing block - block selection bit 1            TrvBit2         : BOOL:=0;              // EPOS-Wort-1 BIT 02 --> 1 = Traversing block - block selection bit 2            TrvBit3         : BOOL:=0;              // EPOS-Wort-1 BIT 03 --> 1 = Traversing block - block selection bit 3            TrvBit4         : BOOL:=0;              // EPOS-Wort-1 BIT 04 --> 1 = Traversing block - block selection bit 4            TrvBit5         : BOOL:=0;              // EPOS-Wort-1 Bit 05 --> 1 = Traversing block - block selection bit 5            Bit06           : BOOL:=0;              // EPOS-Wort-1 Bit 06 --> 1 = Reserve            Bit07           : BOOL:=0;              // EPOS-Wort-1 Bit 07 --> 1 = Reserve          END_STRUCT;
         EPosSTW2 : Word := WORD#16#0000;   // EPOSSTW2sxEPosSTW2   : STRUCT            RefTyp          : BOOL:=0;              // EPOS-Wort-2 Bit 08 --> 1 = Referencing type             RefStDi         : BOOL:=0;              // EPOS-Wort-2 Bit 09 --> 1 = Homing start direction            RefInpS         : BOOL:=0;              // EPOS-Wort-2 Bit 10 --> 1 = Referencing passive - input selection            RefEdge         : BOOL:=0;              // EPOS-Wort-2 Bit 11 --> 1 = Referencing passive - edge evaluation            Bit12           : BOOL:=0;              // EPOS-Wort-2 Bit 12 --> 1 = Reserve            Bit13           : BOOL:=0;              // EPOS-Wort-2 Bit 13 --> 1 = Reserve            SftLimAct       : BOOL:=0;              // EPOS-Wort-2 Bit 14 --> 1 = Software limit switch activation            StpCamAct       : BOOL:=0;              // EPOS-Wort-2 Bit 15 --> 1 = Stop output cam activation            TrkMode         : BOOL:=0;              // EPOS-Wort-2 Bit 00 --> 1 = Tracking mode active            SetRefPt        : BOOL:=0;              // EPOS-Wort-2 Bit 01 --> 1 = Set reference point            ActRefCam       : BOOL:=0;              // EPOS-Wort-2 Bit 02 --> 1 = Reference cam active            Bit03           : BOOL:=0;              // EPOS-Wort-2 Bit 03 --> 1 = Reserve            Bit04           : BOOL:=0;              // EPOS-Wort-2 Bit 04 --> 1 = Reserve            JogInc          : BOOL:=0;              // EPOS-Wort-2 Bit 05 --> 1 = Jogging - jogging incremental            Bit06           : BOOL:=0;              // EPOS-Wort-2 Bit 06 --> 1 = Reserve            Bit07           : BOOL:=0;              // EPOS-Wort-2 Bit 07 --> 1 = Reserve         END_STRUCT;
         STW2 : Word := WORD#16#0000;   // STW2sxSTW2         : STRUCT            TrvFixStp       : BOOL:=0;              // ST-Wort-2 Bit 08 --> 1 = Travel fixed STOP            GlbTrgCom       : BOOL:=0;              // ST-Wort-2 Bit 09 --> 1 = Global trigger command            Bit10           : BOOL:=0;              // ST-Wort-2 Bit 10 --> 1 = Reserve            MotSwOver       : BOOL:=0;              // ST-Wort-2 Bit 11 --> 1 = Motor switch over finished            MsZykBit0       : BOOL:=0;              // ST-Wort-2 Bit 12 --> 1 = Master life bit 0            MsZykBit1       : BOOL:=0;              // ST-Wort-2 Bit 13 --> 1 = Master life bit 1            MsZykBit2       : BOOL:=0;              // ST-Wort-2 Bit 14 --> 1 = Master life bit 2            MsZykBit3       : BOOL:=0;              // ST-Wort-2 Bit 15 --> 1 = Master life bit 3            DDSBit0         : BOOL:=0;              // ST-Wort-2 Bit 00 --> 1 = Drive data set bit 0            DDSBit1         : BOOL:=0;              // ST-Wort-2 Bit 01 --> 1 = Drive data set bit 1            DDSBit2         : BOOL:=0;              // ST-Wort-2 Bit 02 --> 1 = Drive data set bit 2            DDSBit3         : BOOL:=0;              // ST-Wort-2 Bit 03 --> 1 = Drive data set bit 3            DDSBit4         : BOOL:=0;              // ST-Wort-2 Bit 04 --> 1 = Drive data set bit 4            GlbStart        : BOOL:=0;              // ST-Wort-2 Bit 05 --> 1 = Global start            ResIComp        : BOOL:=0;              // ST-Wort-2 Bit 06 --> 1 = Reset I-component of speed controller            ActPrkAxis      : BOOL:=0;              // ST-Wort-2 Bit 07 --> 1 = Activate parking axis            END_STRUCT;
         OverrideV : Word := WORD#16#0000;   // Velocity override
         Position : DWord := DWORD#16#0000_0000;   // Setpoint of position
         Velocity : DWord := DWORD#16#0000_0000;   // Setpoint of velocity
         OverrideA : Word := WORD#16#0000;   // Accelerating override
         OverrideD : Word := WORD#16#0000;   // Decelerating override
         Reserve : Word := WORD#16#0000;   // Reserve
      END_STRUCT;
      sxRecvBuf : Struct   // receive buffer of telegram for receiving data from the drive
         ZSW1 : Word := WORD#16#0000;   // ZSW1sxZSW1         : STRUCT            NoFlwErr        : BOOL:=0;              // ZSW-Wort-1 Bit 08 --> 1 = Following error in tolerance            LbCr            : BOOL:=0;              // ZSW-Wort-1 Bit 09 --> 1 = Lifebit control request            TargPos         : BOOL:=0;              // ZSW-Wort-1 Bit 10 --> 1 = Target position reached            RefPSet         : BOOL:=0;              // ZSW-Wort-1 Bit 11 --> 1 = Reference point set            TrvTskAck       : BOOL:=0;              // ZSW-Wort-1 Bit 12 --> 1 = Traversing task acknowledge            StndStill       : BOOL:=0;              // ZSW-Wort-1 Bit 13 --> 1 = [n_ist] < Drehzahlsollwert 3            Accel           : BOOL:=0;              // ZSW-Wort-1 Bit 14 --> 1 = Axis accelerating            Decel           : BOOL:=0;              // ZSW-Wort-1 Bit 15 --> 1 = Axis decelerating            RTS             : BOOL:=0;              // ZSW-Wort-1 Bit 00 --> 1 = Ready to power up / to start            RDY             : BOOL:=0;              // ZSW-Wort-1 Bit 01 --> 1 = Ready to operate             IOp             : BOOL:=0;              // ZSW-Wort-1 Bit 02 --> 1 = In operation (operation enabled)            Fault           : BOOL:=0;              // ZSW-Wort-1 Bit 03 --> 1 = Fault present            NoOff2Act       : BOOL:=0;              // ZSW-Wort-1 Bit 04 --> 1 = OFF2 inactive            NoOff3Act       : BOOL:=0;              // ZSW-Wort-1 Bit 05 --> 1 = OFF3 inactive            PowInhbt        : BOOL:=0;              // ZSW-Wort-1 Bit 06 --> 1 = Power ON inhibit active             Alarm           : BOOL:=0;              // ZSW-Wort-1 Bit 07 --> 1 = Alarm / Warning present         END_STRUCT;
         EPosZSW1 : Word := WORD#16#0000;   // EPOSZSW1sxEPosZSW1     : STRUCT            StpCamMinAct    : BOOL:=0;              // EPOS-Wort-1 Bit 08 --> 1 = STOP cam minus active            StpCamPlsAct    : BOOL:=0;              // EPOS-Wort-1 Bit 09 --> 1 = STOP cam plus active            JogAct          : BOOL:=0;              // EPOS-Wort-1 Bit 10 --> 1 = Jogging active            RefAct          : BOOL:=0;              // EPOS-Wort-1 Bit 11 --> 1 = Reference point approach active            FlyRefAct       : BOOL:=0;              // EPOS-Wort-1 Bit 12 --> 1 = Flying referencing active            TrvBlAct        : BOOL:=0;              // EPOS-Wort-1 Bit 13 --> 1 = Traversing block active            MdiStupAct      : BOOL:=0;              // EPOS-Wort-1 Bit 14 --> 1 = MDI setup active            MdiPosAct       : BOOL:=0;              // EPOS-Wort-1 Bit 15 --> 1 = MDI positing active            ActTrvBit0      : BOOL:=0;              // EPOS-Wort-1 BIT 00 --> 1 = Active traversing block bit 0            ActTrvBit1      : BOOL:=0;              // EPOS-Wort-1 Bit 01 --> 1 = Active traversing block bit 1            ActTrvBit2      : BOOL:=0;              // EPOS-Wort-1 Bit 02 --> 1 = Active traversing block bit 2            ActTrvBit3      : BOOL:=0;              // EPOS-Wort-1 Bit 03 --> 1 = Active traversing block bit 3            ActTrvBit4      : BOOL:=0;              // EPOS-Wort-1 Bit 04 --> 1 = Active traversing block bit 4            ActTrvBit5      : BOOL:=0;              // EPOS-Wort-1 Bit 05 --> 1 = Active traversing block bit 5            Bit06           : BOOL:=0;              // EPOS-Wort-1 Bit 06 --> 1 = Reserve            Bit07           : BOOL:=0;              // EPOS-Wort-1 Bit 07 --> 1 = Reserve         END_STRUCT;
         EPosZSW2 : Word := WORD#16#0000;   // EPOSZSW2sxEPosZSW2      : STRUCT            PosSmCam1       : BOOL:=0;              // EPOS-Wort-2 Bit 08 --> 1 = Position actual value <= cam position 1            PosSmCam2       : BOOL:=0;              // EPOS-Wort-2 Bit 09 --> 1 = Position actual value <= cam position 2            TrvOut1         : BOOL:=0;              // EPOS-Wort-2 Bit 10 --> 1 = Direct output 1 via traversing block            TrvOut2         : BOOL:=0;              // EPOS-Wort-2 Bit 11 --> 1 = Direct output 2 via traversing block             FxStpRd         : BOOL:=0;              // EPOS-Wort-2 Bit 12 --> 1 = Fixed STOP reached            FxStpTrRd       : BOOL:=0;              // EPOS-Wort-2 Bit 13 --> 1 = Fixed STOP clamping torque reached            TrvFxStpAct     : BOOL:=0;              // EPOS-Wort-2 Bit 14 --> 1 = Traversing fixed STOP active            CmdAct          : BOOL:=0;              // EPOS-Wort-2 Bit 15 --> 1 = Traversing command active            TrkModeAct      : BOOL:=0;              // EPOS-Wort-2 Bit 00 --> 1 = Tracking mode active            VeloLimAct      : BOOL:=0;              // EPOS-Wort-2 Bit 01 --> 1 = Velocity limit active            SetPStat        : BOOL:=0;              // EPOS-Wort-2 Bit 02 --> 1 = Setpoint static            PrnMrkOut       : BOOL:=0;              // EPOS-Wort-2 Bit 03 --> 1 = Printmark outside outer window            FWD             : BOOL:=0;              // EPOS-Wort-2 Bit 04 --> 1 = Axis forwards            BWD             : BOOL:=0;              // EPOS-Wort-2 Bit 05 --> 1 = Axis backwards            SftSwMinAct     : BOOL:=0;              // EPOS-Wort-2 Bit 06 --> 1 = Software limit switch minus active            SftSwPlsAct     : BOOL:=0;              // EPOS-Wort-2 Bit 07 --> 1 = Software limit switch plus active         END_STRUCT;
         ZSW2 : Word := WORD#16#0000;   // ZSW2sxZSW2     : STRUCT            Bit08           : BOOL:=0;              // ZSW-Wort-2 Bit 08 --> Reserve            GlbTrgReq       : BOOL:=0;              // ZSW-Wort-2 Bit 09 --> Global trigger request            PulsEn          : BOOL:=0;              // ZSW-Wort-2 Bit 10 --> Pulses enabled            MotSwOverAct    : BOOL:=0;              // ZSW-Wort-2 Bit 11 --> Motor switch over activ            SlvZykBit0      : BOOL:=0;              // ZSW-Wort-2 Bit 12 --> Slave - life bit 0            SlvZykBit1      : BOOL:=0;              // ZSW-Wort-2 Bit 13 --> Slave - life bit 1            SlvZykBit2      : BOOL:=0;              // ZSW-Wort-2 Bit 14 --> Slave - life bit 2            SlvZykBit3      : BOOL:=0;              // ZSW-Wort-2 Bit 15 --> Slave - life bit 3            ActDDSBit0      : BOOL:=0;              // ZSW-Wort-2 Bit 00 --> Active drive data set bit 0            ActDDSBit1      : BOOL:=0;              // ZSW-Wort-2 Bit 01 --> Active drive data set bit 1            ActDDSBit2      : BOOL:=0;              // ZSW-Wort-2 Bit 02 --> Active drive data set bit 2            ActDDSBit3      : BOOL:=0;              // ZSW-Wort-2 Bit 03 --> Active drive data set bit 3            ActDDSBit4      : BOOL:=0;              // ZSW-Wort-2 Bit 04 --> Active drive data set bit 4            CmdActRelBrk    : BOOL:=0;              // ZSW-Wort-2 Bit 05 --> Command "release holding break" active            TrqContMode     : BOOL:=0;              // ZSW-Wort-2 Bit 06 --> Torque controlled mode            ParkAxisAct     : BOOL:=0;              // ZSW-Wort-2 Bit 07 --> Parking axis activated            END_STRUCT;
         NotUsed : Word := WORD#16#0000;   // Reserve
         Position : DWord := DWORD#16#0000_0000;   // Feedback of position
         Velocity : DWord := DWORD#16#0000_0000;   // Feedback of velocity
         ErrNr : Word := WORD#16#0000;   // Fault number
         WarnNr : Word := WORD#16#0000;   // Warning number
         Reserve : Word := WORD#16#0000;   // Reserve
      END_STRUCT;
   END_VAR

   VAR_TEMP 
      piRetSFC : Int;   // Status for fault analysis
      piCount : Int;   // Freely available counter variable 3
      swSendBuf : Array[0..11] of Word;   // Send buffer
      swRecvBuf : Array[0..11] of Word;   // Receive buffer
   END_VAR


BEGIN
	
	//=============================================================================
	//SIEMENS AG
	//(c)Copyright 2019 All Rights Reserved
	//-----------------------------------------------------------------------------
	// Library: DriveLib
	// Tested with: -
	// Engineering: TIA Portal V15.1
	// Restrictions: -
	// Requirements: S7-1200 / S7-1500
	// Functionality: cyclic communication between a SINAMICS (Basic positioner)and a PLC
	//                If in HWConfig Std.TLG 111 is projected 12 PZD-words are exchanged
	//                in every bus cycle.
	//                The parametrisation of these words is described in the manual of the
	//                SINAMICS
	//=============================================================================
	
	// Betriebsart ermitteln
	IF #ModePos > #siModePosMax THEN
	  
	  #sbModePos := FALSE;
	  #Error := True;
	  #swStatus := 16#8202;
	ELSIF #ModePos < 1 THEN
	  
	  #sbModePos := FALSE;
	  #Error := True;
	  #swStatus := 16#8202;
	ELSE
	  // Betriebsartenwechsel ist nur möglich, wenn die Achse nicht beschleunigt oder nicht verzögert 
	  // und die Geschwindigkeit Null ist
	  IF NOT #sbFWD AND NOT #sbBWD AND NOT #sbAccel AND NOT #sbDecel THEN
	    
	    #sbModePos := TRUE;
	    #siModePos := #ModePos;
	    
	    // Fehler wieder zurücknehmen, wenn er mal ausgelöst wurde
	    IF #swStatus = 16#8202 THEN
	      #swStatus := 16#7002;
	      #Error := False;
	    END_IF;
	  END_IF;
	END_IF;
	
	// Überprüfung der analogen Eingabewerte, ob sie innerhalb des möglichen Bereiches liegen
	// Geschwindigkeitsoverride (0% - 199%, 100% => W#16#4000)
	IF (#OverV < 0) OR (#OverV > 199) THEN
	  #swStatus := 16#8203;
	  #Error := True;
	ELSE
	  // Geschwindigkeitsoverride in den Sendepuffer eintragen
	  #sxSendBuf.OverrideV := INT_TO_WORD(REAL_TO_INT(16384.0 * (INT_TO_REAL(#OverV) / 100.0)));
	END_IF;
	
	// Beschleunigungsoverride (0% - 100%, 100% => W#16#4000)
	IF (#OverAcc < 0) OR (#OverAcc > 100) THEN
	  #swStatus := 16#8203;
	  #Error := True;
	ELSE
	  // Beschleunigungsoverride in den Sendepuffer eintragen
	  #sxSendBuf.OverrideA := INT_TO_WORD(REAL_TO_INT(16384.0 * (INT_TO_REAL(#OverAcc) / 100.0)));
	END_IF;
	
	// Verzögerungsoverride (0% - 100%, 100% => W#16#4000)
	IF (#OverDec < 0) OR (#OverDec > 100) THEN
	  #swStatus := 16#8203;
	  #Error := True;
	ELSE
	  // Verzögerungsoverride in den Sendepuffer eintragen
	  #sxSendBuf.OverrideD := INT_TO_WORD(REAL_TO_INT(16384.0 * (INT_TO_REAL(#OverDec) / 100.0)));
	END_IF;
	
	// Fehler wieder zurücknehmen, wenn er mal ausgelöst wurde
	IF NOT (#OverV < 0) AND NOT (#OverV > 199) AND NOT (#OverAcc < 0) AND NOT (#OverAcc > 100) AND
	  NOT (#OverDec < 0) AND NOT (#OverDec > 100) THEN
	  IF #swStatus = 16#8203 THEN
	    #swStatus := 16#7002;
	    #Error := False;
	  END_IF;
	END_IF;
	
	// Positionssollwert
	// Positionssollwert in den Sendepuffer eintragen
	#sxSendBuf.Position := DINT_TO_DWORD(#Position);
	
	// Geschwindigkeitssollwert (Begrenzung / Überwachung
	// Geschwindigkeitssollwert in den Sendepuffer eintragen
	#sxSendBuf.Velocity := DINT_TO_DWORD(#Velocity);
	
	// Einschalten bzw. Ausschalten des Antriebes erkennen
	IF #EnableAxis AND NOT #sbOff1Edge AND NOT #sbBusy AND #sbModePos THEN
	  #sbOff1 := True;
	END_IF;
	// Einschalten bzw. Ausschalten des Antriebes Flanke merken
	#sbOff1Edge := #EnableAxis AND NOT #sbBusy;
	
	// Einschaltflankenmerker wieder zurücksetzen
	IF NOT #EnableAxis THEN
	  #sbOff1 := False;
	END_IF;
	
	// Fliegendes Referenzieren aktivieren erkennen
	IF #FlyRef AND NOT #sbRefTypEdge THEN
	  #sbRefTyp := True;
	END_IF;
	// Fliegendes Referenzieren aktivieren Flanke merken
	#sbRefTypEdge := #FlyRef;
	
	// Fliegendes Referenzieren Flankenmerker wieder zurücksetzen
	IF NOT #FlyRef THEN
	  #sbRefTyp := False;
	  #siRefTypCyc := 0;
	END_IF;
	
	// Betriebsart aktivieren erkennen (RQ 3901129, RQ 4094299)
	IF #ExecuteMode AND NOT #sbExecuteEdge THEN
	  #sbExecute := True;
	  #siExecuteCyc := 0;
	ELSIF #ActMode <> #ModePos THEN
	  #sbExecute := FALSE;
	ELSIF #siExecuteCyc > (2 * #siCycWait) THEN
	  IF #ModePos <> 4 THEN
	    #sbExecute := FALSE;
	  ELSE
	    IF #sxRecvBuf.ZSW1.%X11 OR NOT #ExecuteMode THEN
	      #sbExecute := FALSE;
	    END_IF;
	  END_IF;
	ELSE
	  ; // not used
	END_IF;
	
	IF #siExecuteCyc > 100 THEN
	  #siExecuteCyc := 0;
	ELSE
	  #siExecuteCyc := #siExecuteCyc + 1;
	END_IF;
	
	// Verfahrauftrag aktivieren Flanke merken
	#sbExecuteEdge := #ExecuteMode;
	
	// Betriebsart MDI / Sollwertdirektvorgabe Flanke merken
	(*IF #sxSendBuf.sxEPosSTW1.MdiStart AND NOT #sbMdiStartEdge THEN
	          #sbMdiStart := True;
	      END_IF;
	      // Betriebsart MDI / Sollwertdirektvorgabe Flanke merken
	      #sbMdiStartEdge := #sxSendBuf.sxEPosSTW1.MdiStart AND NOT #Busy;*)
	
	// Verfahrauftragflankenmerker wieder zurücksetzen
	(*IF NOT #sxSendBuf.sxEPosSTW1.MdiStart THEN
	          #sbMdiStart := False;
	          #siMdiStartCyc := 0;
	      END_IF;*)
	
	IF #sxSendBuf.EPosSTW1.%X15 AND NOT #sbMdiStartEdge THEN
	  #sbMdiStart := True;
	END_IF;
	// Betriebsart MDI / Sollwertdirektvorgabe Flanke merken
	#sbMdiStartEdge := #sxSendBuf.EPosSTW1.%X15 AND NOT #sbBusy;
	
	// Verfahrauftragflankenmerker wieder zurücksetzen
	IF NOT #sxSendBuf.EPosSTW1.%X15 THEN
	  #sbMdiStart := False;
	  #siMdiStartCyc := 0;
	END_IF;
	
	// Schreibdaten zusammenstellen
	// Steuerword STW1 für alle Betriebsart aufbereiten
	(*#sxSendBuf.sxSTW1.RejTrvTsk        := #RejTrvTsk;
	      #sxSendBuf.sxSTW1.IntMStop         := #IntMStop;
	      #sxSendBuf.sxSTW1.AckFault         := #AckFlt;*)
	
	#sxSendBuf.STW1.%X4 := #CancelTraversing;
	#sxSendBuf.STW1.%X5 := #IntermediateStop;
	#sxSendBuf.STW1.%X7 := #AckError;
	#sxSendBuf.STW1.%X1 := TRUE;
	#sxSendBuf.STW1.%X2 := TRUE;
	#sxSendBuf.STW1.%X3 := TRUE;
	#sxSendBuf.STW1.%X10 := TRUE;
	
	// Hauptbetriebsart "Positionieren / manueller Sollwertvorgabe (MDI)" 
	// Betriebsart "Positionieren Relativ positiv" oder "Positionieren Relativ negativ"
	IF (#siModePos = 1 AND #sbModePos) THEN
	  
	  // Antrieb einschalten
	  //#sxSendBuf.sxSTW1.Off1 := #sbOff1;
	  #sxSendBuf.STW1.%X0 := #sbOff1;
	  
	  // nicht verwendete Signale für den 1. Schritt und eventuell weitere Schritte
	  (*#sxSendBuf.sxSTW1.Jog1          := False;
	          #sxSendBuf.sxSTW1.Jog2          := False;
	          #sxSendBuf.sxEPosSTW1.MdiTyp    := False;
	          #sxSendBuf.sxEPosSTW1.MdiPos    := False;
	          #sxSendBuf.sxEPosSTW1.MdiNeg    := False;
	          #sxSendBuf.sxEPosSTW1.MdiSetup  := False;
	          #sxSendBuf.sxEPosSTW2.SetRefPt  := False;
	          #sxSendBuf.sxEPosSTW2.JogInc    := False;
	          #sxSendBuf.sxEPosSTW2.RefStDi   := False;
	          #sxSendBuf.sxSTW1.RefStart      := False;
	          #sxSendBuf.sxEPosSTW2.RefTyp    := False;
	          #sxSendBuf.sxEPosSTW1.MdiStart  := False;*)
	  #sxSendBuf.STW1.%X8 := False;
	  #sxSendBuf.STW1.%X9 := False;
	  #sxSendBuf.EPosSTW1.%X8 := False;
	  #sxSendBuf.EPosSTW1.%X9 := False;
	  #sxSendBuf.EPosSTW1.%X10 := False;
	  #sxSendBuf.EPosSTW1.%X14 := False;
	  #sxSendBuf.EPosSTW2.%X1 := False;
	  #sxSendBuf.EPosSTW2.%X5 := False;
	  #sxSendBuf.EPosSTW2.%X9 := False;
	  #sxSendBuf.STW1.%X11 := False;
	  #sxSendBuf.EPosSTW2.%X8 := False;
	  #sxSendBuf.EPosSTW1.%X15 := False;
	  
	  
	  // Nach dem Einschalten des Antriebes, prüfen ob der Antrieb betriebsbereit, in Operation ohne Fehler und Warnung ist, 
	  // dann die Betriebsart MDI / Sollwertvorgabe Start gesetzt werden
	  IF #sbOff1 AND #sbReady AND #sbIOp AND NOT #sbFault THEN
	    
	    // Betriebsart MDI / Sollwertdirektvorgabe setzen
	    //#sxSendBuf.sxEPosSTW1.MdiStart := True;
	    #sxSendBuf.EPosSTW1.%X15 := True;
	    
	    // Positioniertyp auf relatives Positionieren stellen 
	    //#sxSendBuf.sxEPosSTW1.MdiTyp := False;
	    #sxSendBuf.EPosSTW1.%X8 := False;
	    
	    // die Richtungswahl für das Positionieren auf positive Richtung oder negative Richtung einstellen
	    IF #Positive AND NOT #Negative THEN
	      
	      // positive Richtung
	      //#sxSendBuf.sxEPosSTW1.MdiPos := True;
	      #sxSendBuf.EPosSTW1.%X9 := True;
	      
	      // negative Richtung
	      //#sxSendBuf.sxEPosSTW1.MdiNeg := False;
	      #sxSendBuf.EPosSTW1.%X10 := False;
	      
	      // die Richtungswahl für das Positionieren auf negative Richtung einstellen                
	    ELSIF NOT #Positive AND #Negative THEN
	      
	      // positive Richtung
	      //#sxSendBuf.sxEPosSTW1.MdiPos := False;
	      #sxSendBuf.EPosSTW1.%X9 := False;
	      
	      // negative Richtung
	      //#sxSendBuf.sxEPosSTW1.MdiNeg := True;
	      #sxSendBuf.EPosSTW1.%X10 := True;
	      
	      // die Richtungswahl für das Positionieren auf keine Richtung einstellen                
	    ELSE
	      
	      // positive Richtung
	      //#sxSendBuf.sxEPosSTW1.MdiPos := False;
	      #sxSendBuf.EPosSTW1.%X9 := False;
	      
	      // negative Richtung
	      //#sxSendBuf.sxEPosSTW1.MdiNeg := False;
	      #sxSendBuf.EPosSTW1.%X10 := False;
	      
	    END_IF;
	    
	    // Nach dem Einschalten des Antriebes und dem Betriebsart MDI / Sollwertvorgabe starten, 
	    // ein Paar Zyklen warten bevor die Flanke für die Sollwertübernahme MDI gesetzt werden kann
	    IF #sbMdiStart AND (#siMdiStartCyc < #siCycWait) THEN
	      #siMdiStartCyc := #siMdiStartCyc + 1;
	    ELSE
	      // Flanke Sollwertübernahme MDI
	      //#sxSendBuf.sxSTW1.TrvStart := #Execute;
	      #sxSendBuf.STW1.%X6 := #sbExecute;
	      
	    END_IF;
	    
	    // "Fliegendes Referentieren" aktivieren
	    // "Fliegendes Referenzieren" erst nach Einschalten des Antriebes möglich
	    IF #sbRefTyp THEN
	      
	      // Referenziertyp auf "Fliegendes Referenzieren" einstellen
	      //#sxSendBuf.sxEPosSTW2.RefTyp := True;
	      #sxSendBuf.EPosSTW2.%X8 := True;
	      
	      // Nach der Anwahl des Referenziertyps "Fliegendes Referenzieren", 
	      // ein Zyklus später kann das Referenzieren gestartet
	      IF (#siRefTypCyc = 0) THEN
	        #siRefTypCyc := #siRefTypCyc + 1;
	      ELSE
	        // Referenzieren starten
	        //#sxSendBuf.sxSTW1.RefStart := True;
	        #sxSendBuf.STW1.%X11 := True;
	        
	      END_IF;
	    END_IF;
	  END_IF;
	  
	  // Betriebsart "Positionieren Absolut" oder "Positonieren Absolut positiv" oder "Positionieren Absolut negativ"
	ELSIF #siModePos = 2 AND #sbModePos THEN
	  
	  // Antrieb einschalten
	  //#sxSendBuf.sxSTW1.Off1 := #sbOff1;
	  #sxSendBuf.STW1.%X0 := #sbOff1;
	  
